LIN {X 0,Y 417.442,Z 383.937,A -85,B 0,C 180,E1 -10178.471,E2 -10178.471} C_VEL
LIN {X 0,Y 417.791,Z 376.994,A -85,B 0,C 180,E1 -10179.929,E2 -10179.929} C_VEL
LIN {X 0,Y 418.22,Z 369.9,A -85,B 0,C 180,E1 -10181.142,E2 -10181.142} C_VEL
LIN {X 0,Y 418.782,Z 361.342,A -85,B 0,C 180,E1 -10182.355,E2 -10182.355} C_VEL
LIN {X 0,Y 419.399,Z 350.75,A -85,B 0,C 180,E1 -10183.568,E2 -10183.568} C_VEL
LIN {X 0,Y 420.122,Z 340.277,A -85,B 0,C 180,E1 -10184.532,E2 -10184.532} C_VEL
LIN {X 0,Y 420.811,Z 328.769,A -85,B 0,C 180,E1 -10185.374,E2 -10185.374} C_VEL
LIN {X 0,Y 421.406,Z 316.866,A -85,B 0,C 180,E1 -10186.035,E2 -10186.035} C_VEL
LIN {X 0,Y 422.047,Z 303.154,A -85,B 0,C 180,E1 -10186.569,E2 -10186.569} C_VEL
LIN {X 0,Y 422.362,Z 290.817,A -85,B 0,C 180,E1 -10186.867,E2 -10186.867} C_VEL
LIN {X 0,Y 422.986,Z 214.349,A -85,B 0,C 180,E1 -10188.185,E2 -10188.185} C_VEL
LIN {X 0,Y 419.308,Z 188.077,A -85,B 0,C 180,E1 -10188.791,E2 -10188.791} C_VEL
LIN {X 0,Y 420.32,Z 170.294,A -85,B 0,C 180,E1 -10192.099,E2 -10192.099} C_VEL
LIN {X 0,Y 421.109,Z 156.698,A -85,B 0,C 180,E1 -10194.66,E2 -10194.66} C_VEL
LIN {X 0,Y 419.458,Z 146.94,A -85,B 0,C 180,E1 -10196.628,E2 -10196.628} C_VEL
LIN {X 0,Y 418.334,Z 141.379,A -85,B 0,C 180,E1 -10197.822,E2 -10197.822} C_VEL
LIN {X 0,Y 418.213,Z 141.391,A -85,B 0,C 180,E1 -10201.396,E2 -10201.396} C_VEL
LIN {X 0,Y 418.267,Z 141.381,A -85,B 0,C 180,E1 -10204.58,E2 -10204.58} C_VEL
LIN {X 0,Y 418.231,Z 141.391,A -85,B 0,C 180,E1 -10207.833,E2 -10207.833} C_VEL
LIN {X 0,Y 418.224,Z 141.385,A -85,B 0,C 180,E1 -10210.948,E2 -10210.948} C_VEL
LIN {X 0,Y 418.211,Z 141.394,A -85,B 0,C 180,E1 -10213.729,E2 -10213.729} C_VEL
LIN {X 0,Y 418.209,Z 141.387,A -85,B 0,C 180,E1 -10216.448,E2 -10216.448} C_VEL
LIN {X 0,Y 418.223,Z 141.387,A -85,B 0,C 180,E1 -10219.13,E2 -10219.13} C_VEL
LIN {X 0,Y 418.226,Z 141.386,A -85,B 0,C 180,E1 -10222.167,E2 -10222.167} C_VEL
LIN {X 0,Y 418.264,Z 141.387,A -85,B 0,C 180,E1 -10225.42,E2 -10225.42} C_VEL
LIN {X 0,Y 418.211,Z 141.387,A -85,B 0,C 180,E1 -10228.604,E2 -10228.604} C_VEL
LIN {X 0,Y 418.292,Z 141.378,A -85,B 0,C 180,E1 -10231.936,E2 -10231.936} C_VEL
LIN {X 0,Y 418.29,Z 141.383,A -85,B 0,C 180,E1 -10235.162,E2 -10235.162} C_VEL
LIN {X 0,Y 418.234,Z 141.384,A -85,B 0,C 180,E1 -10238.303,E2 -10238.303} C_VEL
LIN {X 0,Y 418.276,Z 141.383,A -85,B 0,C 180,E1 -10241.383,E2 -10241.383} C_VEL
LIN {X 0,Y 418.302,Z 141.376,A -85,B 0,C 180,E1 -10244.406,E2 -10244.406} C_VEL
LIN {X 0,Y 418.355,Z 141.371,A -85,B 0,C 180,E1 -10247.385,E2 -10247.385} C_VEL
LIN {X 0,Y 418.339,Z 141.372,A -85,B 0,C 180,E1 -10250.328,E2 -10250.328} C_VEL
LIN {X 0,Y 418.46,Z 141.358,A -85,B 0,C 180,E1 -10253.248,E2 -10253.248} C_VEL
LIN {X 0,Y 418.336,Z 141.374,A -85,B 0,C 180,E1 -10255.181,E2 -10255.181} C_VEL
LIN {X 0,Y 418.543,Z 141.346,A -85,B 0,C 180,E1 -10258.075,E2 -10258.075} C_VEL
LIN {X 0,Y 418.671,Z 141.33,A -85,B 0,C 180,E1 -10260,E2 -10260} C_VEL
LIN {X 0,Y 418.508,Z 141.354,A -85,B 0,C 180,E1 -10262.888,E2 -10262.888} C_VEL
LIN {X 0,Y 418.487,Z 141.357,A -85,B 0,C 180,E1 -10266.751,E2 -10266.751} C_VEL
LIN {X 0,Y 418.34,Z 141.371,A -85,B 0,C 180,E1 -10269.671,E2 -10269.671} C_VEL
LIN {X 0,Y 418.346,Z 141.371,A -85,B 0,C 180,E1 -10273.001,E2 -10273.001} C_VEL
LIN {X 0,Y 418.312,Z 141.377,A -85,B 0,C 180,E1 -10276.735,E2 -10276.735} C_VEL
LIN {X 0,Y 418.27,Z 141.382,A -85,B 0,C 180,E1 -10279.79,E2 -10279.79} C_VEL
LIN {X 0,Y 418.231,Z 141.386,A -85,B 0,C 180,E1 -10282.736,E2 -10282.736} C_VEL
LIN {X 0,Y 418.267,Z 141.385,A -85,B 0,C 180,E1 -10285.904,E2 -10285.904} C_VEL
LIN {X 0,Y 418.264,Z 141.38,A -85,B 0,C 180,E1 -10289.162,E2 -10289.162} C_VEL
LIN {X 0,Y 418.256,Z 141.381,A -85,B 0,C 180,E1 -10292.844,E2 -10292.844} C_VEL
LIN {X 0,Y 418.244,Z 141.386,A -85,B 0,C 180,E1 -10296.238,E2 -10296.238} C_VEL
LIN {X 0,Y 418.253,Z 141.388,A -85,B 0,C 180,E1 -10299.681,E2 -10299.681} C_VEL
LIN {X 0,Y 418.229,Z 141.386,A -85,B 0,C 180,E1 -10302.321,E2 -10302.321} C_VEL
LIN {X 0,Y 418.234,Z 141.385,A -85,B 0,C 180,E1 -10305.109,E2 -10305.109} C_VEL
LIN {X 0,Y 418.239,Z 141.389,A -85,B 0,C 180,E1 -10307.767,E2 -10307.767} C_VEL
LIN {X 0,Y 418.244,Z 141.383,A -85,B 0,C 180,E1 -10310.621,E2 -10310.621} C_VEL
LIN {X 0,Y 418.241,Z 141.385,A -85,B 0,C 180,E1 -10313.976,E2 -10313.976} C_VEL
LIN {X 0,Y 418.256,Z 141.386,A -85,B 0,C 180,E1 -10317.156,E2 -10317.156} C_VEL
LIN {X 0,Y 418.268,Z 141.382,A -85,B 0,C 180,E1 -10320.896,E2 -10320.896} C_VEL
LIN {X 0,Y 418.268,Z 141.38,A -85,B 0,C 180,E1 -10324.096,E2 -10324.096} C_VEL
LIN {X 0,Y 418.232,Z 141.39,A -85,B 0,C 180,E1 -10327.264,E2 -10327.264} C_VEL
LIN {X 0,Y 418.282,Z 141.378,A -85,B 0,C 180,E1 -10330.364,E2 -10330.364} C_VEL
LIN {X 0,Y 418.316,Z 141.376,A -85,B 0,C 180,E1 -10333.405,E2 -10333.405} C_VEL
LIN {X 0,Y 418.346,Z 141.377,A -85,B 0,C 180,E1 -10336.999,E2 -10336.999} C_VEL
LIN {X 0,Y 418.339,Z 141.372,A -85,B 0,C 180,E1 -10340.329,E2 -10340.329} C_VEL
LIN {X 0,Y 418.46,Z 141.358,A -85,B 0,C 180,E1 -10343.249,E2 -10343.249} C_VEL
LIN {X 0,Y 418.336,Z 141.377,A -85,B 0,C 180,E1 -10345.182,E2 -10345.182} C_VEL
LIN {X 0,Y 418.543,Z 141.351,A -85,B 0,C 180,E1 -10348.076,E2 -10348.076} C_VEL
LIN {X 0,Y 418.534,Z 141.54,A -85,B 0,C 180,E1 -10348.797,E2 -10348.797} C_VEL
LIN {X 0,Y 419.76,Z 148.679,A -85,B 0,C 180,E1 -10350.48,E2 -10350.48} C_VEL
LIN {X 0,Y 419.846,Z 152.338,A -85,B 0,C 180,E1 -10351.31,E2 -10351.31} C_VEL
LIN {X 0,Y 423.514,Z 171.824,A -85,B 0,C 180,E1 -10351.804,E2 -10351.804} C_VEL
LIN {X 0,Y 423.009,Z 213.686,A -85,B 0,C 180,E1 -10352.52,E2 -10352.52} C_VEL
LIN {X 0,Y 422.295,Z 219.534,A -85,B 0,C 180,E1 -10352.597,E2 -10352.597} C_VEL
LIN {X 0,Y 416.394,Z 238.495,A -85,B 0,C 180,E1 -10352.713,E2 -10352.713} C_VEL
LIN {X 0,Y 415.758,Z 244.339,A -85,B 0,C 180,E1 -10352.794,E2 -10352.794} C_VEL
LIN {X 0,Y 415.479,Z 262.827,A -85,B 0,C 180,E1 -10353.167,E2 -10353.167} C_VEL
LIN {X 0,Y 415.18,Z 275.079,A -85,B 0,C 180,E1 -10353.598,E2 -10353.598} C_VEL
LIN {X 0,Y 414.746,Z 286.827,A -85,B 0,C 180,E1 -10354.191,E2 -10354.191} C_VEL
LIN {X 0,Y 414.175,Z 298.648,A -85,B 0,C 180,E1 -10354.989,E2 -10354.989} C_VEL
LIN {X 0,Y 413.529,Z 310.039,A -85,B 0,C 180,E1 -10355.975,E2 -10355.975} C_VEL
LIN {X 0,Y 412.809,Z 320.326,A -85,B 0,C 180,E1 -10357.09,E2 -10357.09} C_VEL
LIN {X 0,Y 412.06,Z 330.114,A -85,B 0,C 180,E1 -10358.416,E2 -10358.416} C_VEL
LIN {X 0,Y 411.453,Z 338.576,A -85,B 0,C 180,E1 -10359.835,E2 -10359.835} C_VEL
LIN {X 0,Y 410.99,Z 345.766,A -85,B 0,C 180,E1 -10361.341,E2 -10361.341} C_VEL
LIN {X 0,Y 410.619,Z 351.496,A -85,B 0,C 180,E1 -10362.856,E2 -10362.856} C_VEL
LIN {X 0,Y 410.329,Z 355.996,A -85,B 0,C 180,E1 -10364.38,E2 -10364.38} C_VEL
LIN {X 0,Y 410.103,Z 359.379,A -85,B 0,C 180,E1 -10365.914,E2 -10365.914} C_VEL
LIN {X 0,Y 409.981,Z 361.058,A -85,B 0,C 180,E1 -10366.943,E2 -10366.943} C_VEL
LIN {X 0,Y 409.908,Z 362.294,A -85,B 0,C 180,E1 -10367.976,E2 -10367.976} C_VEL
LIN {X 0,Y 409.918,Z 363.263,A -85,B 0,C 180,E1 -10369.444,E2 -10369.444} C_VEL
LIN {X 0,Y 409.88,Z 363.307,A -85,B 0,C 180,E1 -10371.105,E2 -10371.105} C_VEL
LIN {X 0,Y 409.945,Z 362.679,A -85,B 0,C 180,E1 -10372.217,E2 -10372.217} C_VEL
LIN {X 0,Y 410.041,Z 361.707,A -85,B 0,C 180,E1 -10373.217,E2 -10373.217} C_VEL
LIN {X 0,Y 410.288,Z 359.319,A -85,B 0,C 180,E1 -10374.789,E2 -10374.789} C_VEL
LIN {X 0,Y 410.566,Z 355.675,A -85,B 0,C 180,E1 -10376.428,E2 -10376.428} C_VEL
LIN {X 0,Y 410.96,Z 350.746,A -85,B 0,C 180,E1 -10378.053,E2 -10378.053} C_VEL
LIN {X 0,Y 411.519,Z 344.278,A -85,B 0,C 180,E1 -10379.688,E2 -10379.688} C_VEL
LIN {X 0,Y 412.226,Z 336.472,A -85,B 0,C 180,E1 -10381.248,E2 -10381.248} C_VEL
LIN {X 0,Y 413.047,Z 327.312,A -85,B 0,C 180,E1 -10382.699,E2 -10382.699} C_VEL
LIN {X 0,Y 413.821,Z 317.593,A -85,B 0,C 180,E1 -10383.941,E2 -10383.941} C_VEL
LIN {X 0,Y 414.737,Z 306.944,A -85,B 0,C 180,E1 -10385.032,E2 -10385.032} C_VEL
LIN {X 0,Y 415.542,Z 296.131,A -85,B 0,C 180,E1 -10385.91,E2 -10385.91} C_VEL
LIN {X 0,Y 416.147,Z 283.863,A -85,B 0,C 180,E1 -10386.686,E2 -10386.686} C_VEL
LIN {X 0,Y 416.694,Z 271.1,A -85,B 0,C 180,E1 -10387.272,E2 -10387.272} C_VEL
LIN {X 0,Y 417.018,Z 257.825,A -85,B 0,C 180,E1 -10387.664,E2 -10387.664} C_VEL
LIN {X 0,Y 418.238,Z 172.5,A -85,B 0,C 180,E1 -10389.181,E2 -10389.181} C_VEL
LIN {X 0,Y 414.446,Z 156.312,A -85,B 0,C 180,E1 -10389.696,E2 -10389.696} C_VEL
LIN {X 0,Y 413.397,Z 153.147,A -85,B 0,C 180,E1 -10389.83,E2 -10389.83} C_VEL
LIN {X 0,Y 411.182,Z 142.299,A -85,B 0,C 180,E1 -10392.548,E2 -10392.548} C_VEL
LIN {X 0,Y 411.164,Z 142.275,A -85,B 0,C 180,E1 -10395.882,E2 -10395.882} C_VEL
LIN {X 0,Y 411.158,Z 142.269,A -85,B 0,C 180,E1 -10399.493,E2 -10399.493} C_VEL
LIN {X 0,Y 411.186,Z 142.266,A -85,B 0,C 180,E1 -10402.026,E2 -10402.026} C_VEL
LIN {X 0,Y 411.203,Z 142.267,A -85,B 0,C 180,E1 -10405.124,E2 -10405.124} C_VEL
LIN {X 0,Y 411.16,Z 142.269,A -85,B 0,C 180,E1 -10408.002,E2 -10408.002} C_VEL
LIN {X 0,Y 411.17,Z 142.267,A -85,B 0,C 180,E1 -10411.407,E2 -10411.407} C_VEL
LIN {X 0,Y 411.187,Z 142.268,A -85,B 0,C 180,E1 -10414.942,E2 -10414.942} C_VEL
LIN {X 0,Y 411.196,Z 142.259,A -85,B 0,C 180,E1 -10417.913,E2 -10417.913} C_VEL
LIN {X 0,Y 411.178,Z 142.262,A -85,B 0,C 180,E1 -10421.049,E2 -10421.049} C_VEL
LIN {X 0,Y 411.195,Z 142.264,A -85,B 0,C 180,E1 -10424.13,E2 -10424.13} C_VEL
LIN {X 0,Y 411.296,Z 142.25,A -85,B 0,C 180,E1 -10427.166,E2 -10427.166} C_VEL
LIN {X 0,Y 411.274,Z 142.252,A -85,B 0,C 180,E1 -10430.161,E2 -10430.161} C_VEL
LIN {X 0,Y 411.391,Z 142.232,A -85,B 0,C 180,E1 -10433.132,E2 -10433.132} C_VEL
LIN {X 0,Y 411.284,Z 142.249,A -85,B 0,C 180,E1 -10435.099,E2 -10435.099} C_VEL
LIN {X 0,Y 411.502,Z 142.22,A -85,B 0,C 180,E1 -10438.043,E2 -10438.043} C_VEL
LIN {X 0,Y 411.377,Z 142.238,A -85,B 0,C 180,E1 -10440.979,E2 -10440.979} C_VEL
LIN {X 0,Y 411.428,Z 142.225,A -85,B 0,C 180,E1 -10442.938,E2 -10442.938} C_VEL
LIN {X 0,Y 411.429,Z 142.235,A -85,B 0,C 180,E1 -10445.883,E2 -10445.883} C_VEL
LIN {X 0,Y 411.312,Z 142.243,A -85,B 0,C 180,E1 -10448.846,E2 -10448.846} C_VEL
LIN {X 0,Y 411.284,Z 142.248,A -85,B 0,C 180,E1 -10451.833,E2 -10451.833} C_VEL
LIN {X 0,Y 411.256,Z 142.254,A -85,B 0,C 180,E1 -10454.853,E2 -10454.853} C_VEL
LIN {X 0,Y 411.245,Z 142.251,A -85,B 0,C 180,E1 -10457.916,E2 -10457.916} C_VEL
LIN {X 0,Y 411.198,Z 142.264,A -85,B 0,C 180,E1 -10461.034,E2 -10461.034} C_VEL
LIN {X 0,Y 411.219,Z 142.258,A -85,B 0,C 180,E1 -10464.216,E2 -10464.216} C_VEL
LIN {X 0,Y 411.181,Z 142.265,A -85,B 0,C 180,E1 -10467.484,E2 -10467.484} C_VEL
LIN {X 0,Y 411.199,Z 142.259,A -85,B 0,C 180,E1 -10469.713,E2 -10469.713} C_VEL
LIN {X 0,Y 411.209,Z 142.261,A -85,B 0,C 180,E1 -10473.156,E2 -10473.156} C_VEL
LIN {X 0,Y 411.194,Z 142.267,A -85,B 0,C 180,E1 -10476.552,E2 -10476.552} C_VEL
LIN {X 0,Y 411.18,Z 142.265,A -85,B 0,C 180,E1 -10479.722,E2 -10479.722} C_VEL
LIN {X 0,Y 411.172,Z 142.267,A -85,B 0,C 180,E1 -10483.134,E2 -10483.134} C_VEL
LIN {X 0,Y 411.17,Z 142.268,A -85,B 0,C 180,E1 -10485.881,E2 -10485.881} C_VEL
LIN {X 0,Y 411.163,Z 142.272,A -85,B 0,C 180,E1 -10488.772,E2 -10488.772} C_VEL
LIN {X 0,Y 411.192,Z 142.262,A -85,B 0,C 180,E1 -10492.026,E2 -10492.026} C_VEL
LIN {X 0,Y 411.208,Z 142.259,A -85,B 0,C 180,E1 -10495.666,E2 -10495.666} C_VEL
LIN {X 0,Y 411.192,Z 142.268,A -85,B 0,C 180,E1 -10499.152,E2 -10499.152} C_VEL
LIN {X 0,Y 411.255,Z 142.294,A -85,B 0,C 180,E1 -10501.05,E2 -10501.05} C_VEL
LIN {X 0,Y 413.993,Z 154.656,A -85,B 0,C 180,E1 -10503.808,E2 -10503.808} C_VEL
LIN {X 0,Y 414.854,Z 159.972,A -85,B 0,C 180,E1 -10504.943,E2 -10504.943} C_VEL
LIN {X 0,Y 413.792,Z 174.576,A -85,B 0,C 180,E1 -10507.796,E2 -10507.796} C_VEL
LIN {X 0,Y 412.989,Z 187.099,A -85,B 0,C 180,E1 -10510.206,E2 -10510.206} C_VEL
LIN {X 0,Y 417.154,Z 211.973,A -85,B 0,C 180,E1 -10510.896,E2 -10510.896} C_VEL
LIN {X 0,Y 417.661,Z 218.162,A -85,B 0,C 180,E1 -10511.037,E2 -10511.037} C_VEL
LIN {X 0,Y 416.649,Z 296.536,A -85,B 0,C 180,E1 -10512.451,E2 -10512.451} C_VEL
LIN {X 0,Y 416.008,Z 309.504,A -85,B 0,C 180,E1 -10512.867,E2 -10512.867} C_VEL
LIN {X 0,Y 415.3,Z 322.073,A -85,B 0,C 180,E1 -10513.47,E2 -10513.47} C_VEL
LIN {X 0,Y 414.419,Z 334.091,A -85,B 0,C 180,E1 -10514.256,E2 -10514.256} C_VEL
LIN {X 0,Y 413.529,Z 345.578,A -85,B 0,C 180,E1 -10515.231,E2 -10515.231} C_VEL
LIN {X 0,Y 412.662,Z 355.955,A -85,B 0,C 180,E1 -10516.331,E2 -10516.331} C_VEL
LIN {X 0,Y 412.017,Z 364.46,A -85,B 0,C 180,E1 -10517.439,E2 -10517.439} C_VEL
LIN {X 0,Y 411.217,Z 373.705,A -85,B 0,C 180,E1 -10518.914,E2 -10518.914} C_VEL
LIN {X 0,Y 410.654,Z 381.157,A -85,B 0,C 180,E1 -10520.394,E2 -10520.394} C_VEL
LIN {X 0,Y 410.266,Z 388.053,A -85,B 0,C 180,E1 -10522.123,E2 -10522.123} C_VEL
LIN {X 0,Y 410.044,Z 393.055,A -85,B 0,C 180,E1 -10523.775,E2 -10523.775} C_VEL
LIN {X 0,Y 410.009,Z 396.102,A -85,B 0,C 180,E1 -10525.083,E2 -10525.083} C_VEL
LIN {X 0,Y 409.971,Z 399.185,A -85,B 0,C 180,E1 -10527.052,E2 -10527.052} C_VEL
LIN {X 0,Y 410.019,Z 400.129,A -85,B 0,C 180,E1 -10528.035,E2 -10528.035} C_VEL
LIN {X 0,Y 409.982,Z 400.664,A -85,B 0,C 180,E1 -10529.018,E2 -10529.018} C_VEL
LIN {X 0,Y 409.979,Z 400.766,A -85,B 0,C 180,E1 -10530,E2 -10530} C_VEL
LIN {X 0,Y 410.021,Z 399.803,A -85,B 0,C 180,E1 -10531.964,E2 -10531.964} C_VEL
LIN {X 0,Y 409.99,Z 398.717,A -85,B 0,C 180,E1 -10532.948,E2 -10532.948} C_VEL
LIN {X 0,Y 409.944,Z 397.171,A -85,B 0,C 180,E1 -10533.932,E2 -10533.932} C_VEL
LIN {X 0,Y 409.997,Z 394.061,A -85,B 0,C 180,E1 -10535.41,E2 -10535.41} C_VEL
LIN {X 0,Y 410.078,Z 389.873,A -85,B 0,C 180,E1 -10536.89,E2 -10536.89} C_VEL
LIN {X 0,Y 410.368,Z 383.477,A -85,B 0,C 180,E1 -10538.618,E2 -10538.618} C_VEL
LIN {X 0,Y 410.731,Z 376.502,A -85,B 0,C 180,E1 -10540.101,E2 -10540.101} C_VEL
LIN {X 0,Y 411.323,Z 367.744,A -85,B 0,C 180,E1 -10541.581,E2 -10541.581} C_VEL
LIN {X 0,Y 411.907,Z 358.756,A -85,B 0,C 180,E1 -10542.815,E2 -10542.815} C_VEL
LIN {X 0,Y 412.523,Z 348.873,A -85,B 0,C 180,E1 -10543.924,E2 -10543.924} C_VEL
LIN {X 0,Y 413.3,Z 338.012,A -85,B 0,C 180,E1 -10544.903,E2 -10544.903} C_VEL
LIN {X 0,Y 414.029,Z 325.801,A -85,B 0,C 180,E1 -10545.759,E2 -10545.759} C_VEL
LIN {X 0,Y 414.709,Z 313.047,A -85,B 0,C 180,E1 -10546.427,E2 -10546.427} C_VEL
LIN {X 0,Y 415.307,Z 300.463,A -85,B 0,C 180,E1 -10546.877,E2 -10546.877} C_VEL
LIN {X 0,Y 415.557,Z 284.461,A -85,B 0,C 180,E1 -10547.215,E2 -10547.215} C_VEL
LIN {X 0,Y 416.168,Z 215.226,A -85,B 0,C 180,E1 -10548.426,E2 -10548.426} C_VEL
LIN {X 0,Y 412.372,Z 187.703,A -85,B 0,C 180,E1 -10549.087,E2 -10549.087} C_VEL
LIN {X 0,Y 413.612,Z 167.046,A -85,B 0,C 180,E1 -10553.005,E2 -10553.005} C_VEL
LIN {X 0,Y 414.141,Z 157.479,A -85,B 0,C 180,E1 -10554.835,E2 -10554.835} C_VEL
LIN {X 0,Y 411.825,Z 144.813,A -85,B 0,C 180,E1 -10557.45,E2 -10557.45} C_VEL
LIN {X 0,Y 411.29,Z 142.256,A -85,B 0,C 180,E1 -10558.028,E2 -10558.028} C_VEL
LIN {X 0,Y 411.184,Z 142.267,A -85,B 0,C 180,E1 -10561.283,E2 -10561.283} C_VEL
LIN {X 0,Y 411.207,Z 142.262,A -85,B 0,C 180,E1 -10564.333,E2 -10564.333} C_VEL
LIN {X 0,Y 411.198,Z 142.266,A -85,B 0,C 180,E1 -10567.973,E2 -10567.973} C_VEL
LIN {X 0,Y 411.184,Z 142.263,A -85,B 0,C 180,E1 -10570.504,E2 -10570.504} C_VEL
LIN {X 0,Y 411.174,Z 142.264,A -85,B 0,C 180,E1 -10573.133,E2 -10573.133} C_VEL
LIN {X 0,Y 411.168,Z 142.269,A -85,B 0,C 180,E1 -10575.881,E2 -10575.881} C_VEL
LIN {X 0,Y 411.164,Z 142.265,A -85,B 0,C 180,E1 -10578.771,E2 -10578.771} C_VEL
LIN {X 0,Y 411.192,Z 142.263,A -85,B 0,C 180,E1 -10582.026,E2 -10582.026} C_VEL
LIN {X 0,Y 411.205,Z 142.264,A -85,B 0,C 180,E1 -10585.666,E2 -10585.666} C_VEL
LIN {X 0,Y 411.19,Z 142.266,A -85,B 0,C 180,E1 -10589.152,E2 -10589.152} C_VEL
LIN {X 0,Y 411.259,Z 142.253,A -85,B 0,C 180,E1 -10592.522,E2 -10592.522} C_VEL
LIN {X 0,Y 411.22,Z 142.259,A -85,B 0,C 180,E1 -10595.784,E2 -10595.784} C_VEL
LIN {X 0,Y 411.197,Z 142.265,A -85,B 0,C 180,E1 -10598.966,E2 -10598.966} C_VEL
LIN {X 0,Y 411.246,Z 142.254,A -85,B 0,C 180,E1 -10602.084,E2 -10602.084} C_VEL
LIN {X 0,Y 411.26,Z 142.258,A -85,B 0,C 180,E1 -10605.147,E2 -10605.147} C_VEL
LIN {X 0,Y 411.284,Z 142.25,A -85,B 0,C 180,E1 -10608.167,E2 -10608.167} C_VEL
LIN {X 0,Y 411.319,Z 142.249,A -85,B 0,C 180,E1 -10611.154,E2 -10611.154} C_VEL
LIN {X 0,Y 411.444,Z 142.23,A -85,B 0,C 180,E1 -10614.117,E2 -10614.117} C_VEL
LIN {X 0,Y 411.512,Z 142.222,A -85,B 0,C 180,E1 -10618.042,E2 -10618.042} C_VEL
LIN {X 0,Y 411.64,Z 142.206,A -85,B 0,C 180,E1 -10620,E2 -10620} C_VEL
LIN {X 0,Y 411.464,Z 142.231,A -85,B 0,C 180,E1 -10622.937,E2 -10622.937} C_VEL
LIN {X 0,Y 411.451,Z 142.232,A -85,B 0,C 180,E1 -10626.867,E2 -10626.867} C_VEL
LIN {X 0,Y 411.292,Z 142.25,A -85,B 0,C 180,E1 -10629.839,E2 -10629.839} C_VEL
LIN {X 0,Y 411.305,Z 142.248,A -85,B 0,C 180,E1 -10633.104,E2 -10633.104} C_VEL
LIN {X 0,Y 411.257,Z 142.254,A -85,B 0,C 180,E1 -10636.889,E2 -10636.889} C_VEL
LIN {X 0,Y 411.23,Z 142.261,A -85,B 0,C 180,E1 -10639.987,E2 -10639.987} C_VEL
LIN {X 0,Y 411.195,Z 142.261,A -85,B 0,C 180,E1 -10643.148,E2 -10643.148} C_VEL
LIN {X 0,Y 411.236,Z 142.259,A -85,B 0,C 180,E1 -10646.381,E2 -10646.381} C_VEL
LIN {X 0,Y 411.199,Z 142.264,A -85,B 0,C 180,E1 -10649.713,E2 -10649.713} C_VEL
LIN {X 0,Y 411.205,Z 142.26,A -85,B 0,C 180,E1 -10653.156,E2 -10653.156} C_VEL
LIN {X 0,Y 411.191,Z 142.262,A -85,B 0,C 180,E1 -10656.553,E2 -10656.553} C_VEL
LIN {X 0,Y 411.217,Z 142.265,A -85,B 0,C 180,E1 -10659.729,E2 -10659.729} C_VEL
LIN {X 0,Y 411.172,Z 142.265,A -85,B 0,C 180,E1 -10663.134,E2 -10663.134} C_VEL
LIN {X 0,Y 411.166,Z 142.269,A -85,B 0,C 180,E1 -10665.881,E2 -10665.881} C_VEL
LIN {X 0,Y 411.162,Z 142.265,A -85,B 0,C 180,E1 -10668.772,E2 -10668.772} C_VEL
LIN {X 0,Y 411.19,Z 142.263,A -85,B 0,C 180,E1 -10672.026,E2 -10672.026} C_VEL
LIN {X 0,Y 411.203,Z 142.264,A -85,B 0,C 180,E1 -10675.666,E2 -10675.666} C_VEL
LIN {X 0,Y 411.189,Z 142.266,A -85,B 0,C 180,E1 -10679.153,E2 -10679.153} C_VEL
LIN {X 0,Y 411.258,Z 142.253,A -85,B 0,C 180,E1 -10682.522,E2 -10682.522} C_VEL
LIN {X 0,Y 411.219,Z 142.259,A -85,B 0,C 180,E1 -10685.784,E2 -10685.784} C_VEL
LIN {X 0,Y 411.196,Z 142.266,A -85,B 0,C 180,E1 -10688.966,E2 -10688.966} C_VEL
LIN {X 0,Y 411.245,Z 142.255,A -85,B 0,C 180,E1 -10692.085,E2 -10692.085} C_VEL
LIN {X 0,Y 411.259,Z 142.258,A -85,B 0,C 180,E1 -10695.148,E2 -10695.148} C_VEL
LIN {X 0,Y 411.283,Z 142.25,A -85,B 0,C 180,E1 -10698.167,E2 -10698.167} C_VEL
LIN {X 0,Y 411.319,Z 142.249,A -85,B 0,C 180,E1 -10701.154,E2 -10701.154} C_VEL
LIN {X 0,Y 411.444,Z 142.231,A -85,B 0,C 180,E1 -10704.118,E2 -10704.118} C_VEL
LIN {X 0,Y 411.512,Z 142.227,A -85,B 0,C 180,E1 -10708.043,E2 -10708.043} C_VEL
LIN {X 0,Y 411.489,Z 142.365,A -85,B 0,C 180,E1 -10708.593,E2 -10708.593} C_VEL
LIN {X 0,Y 412.843,Z 150.275,A -85,B 0,C 180,E1 -10710.488,E2 -10710.488} C_VEL
LIN {X 0,Y 412.928,Z 152.724,A -85,B 0,C 180,E1 -10711.032,E2 -10711.032} C_VEL
LIN {X 0,Y 416.688,Z 173.001,A -85,B 0,C 180,E1 -10711.555,E2 -10711.555} C_VEL
LIN {X 0,Y 415.758,Z 244.339,A -85,B 0,C 180,E1 -10712.794,E2 -10712.794} C_VEL
LIN {X 0,Y 415.439,Z 248.253,A -85,B 0,C 180,E1 -10712.85,E2 -10712.85} C_VEL
LIN {X 0,Y 413.316,Z 255.899,A -85,B 0,C 180,E1 -10712.913,E2 -10712.913} C_VEL
LIN {X 0,Y 409.135,Z 268.076,A -85,B 0,C 180,E1 -10713.1,E2 -10713.1} C_VEL
LIN {X 0,Y 408.368,Z 272.839,A -85,B 0,C 180,E1 -10713.253,E2 -10713.253} C_VEL
LIN {X 0,Y 408.312,Z 274.666,A -85,B 0,C 180,E1 -10713.329,E2 -10713.329} C_VEL
LIN {X 0,Y 407.854,Z 286.988,A -85,B 0,C 180,E1 -10713.953,E2 -10713.953} C_VEL
LIN {X 0,Y 407.295,Z 298.053,A -85,B 0,C 180,E1 -10714.702,E2 -10714.702} C_VEL
LIN {X 0,Y 406.62,Z 309.609,A -85,B 0,C 180,E1 -10715.704,E2 -10715.704} C_VEL
LIN {X 0,Y 405.886,Z 320.05,A -85,B 0,C 180,E1 -10716.837,E2 -10716.837} C_VEL
LIN {X 0,Y 405.21,Z 328.586,A -85,B 0,C 180,E1 -10717.976,E2 -10717.976} C_VEL
LIN {X 0,Y 404.633,Z 336.423,A -85,B 0,C 180,E1 -10719.245,E2 -10719.245} C_VEL
LIN {X 0,Y 404.072,Z 344.087,A -85,B 0,C 180,E1 -10720.776,E2 -10720.776} C_VEL
LIN {X 0,Y 403.633,Z 350.609,A -85,B 0,C 180,E1 -10722.417,E2 -10722.417} C_VEL
LIN {X 0,Y 403.299,Z 355.81,A -85,B 0,C 180,E1 -10724.121,E2 -10724.121} C_VEL
LIN {X 0,Y 403.053,Z 359.334,A -85,B 0,C 180,E1 -10725.681,E2 -10725.681} C_VEL
LIN {X 0,Y 402.863,Z 361.808,A -85,B 0,C 180,E1 -10727.252,E2 -10727.252} C_VEL
LIN {X 0,Y 402.803,Z 362.878,A -85,B 0,C 180,E1 -10728.304,E2 -10728.304} C_VEL
LIN {X 0,Y 402.822,Z 363.626,A -85,B 0,C 180,E1 -10729.588,E2 -10729.588} C_VEL
LIN {X 0,Y 402.829,Z 363.485,A -85,B 0,C 180,E1 -10731.493,E2 -10731.493} C_VEL
LIN {X 0,Y 402.879,Z 362.797,A -85,B 0,C 180,E1 -10732.568,E2 -10732.568} C_VEL
LIN {X 0,Y 403.033,Z 361.643,A -85,B 0,C 180,E1 -10733.645,E2 -10733.645} C_VEL
LIN {X 0,Y 403.262,Z 359.485,A -85,B 0,C 180,E1 -10735.008,E2 -10735.008} C_VEL
LIN {X 0,Y 403.492,Z 356.523,A -85,B 0,C 180,E1 -10736.37,E2 -10736.37} C_VEL
LIN {X 0,Y 403.892,Z 351.785,A -85,B 0,C 180,E1 -10738.023,E2 -10738.023} C_VEL
LIN {X 0,Y 404.484,Z 345.544,A -85,B 0,C 180,E1 -10739.685,E2 -10739.685} C_VEL
LIN {X 0,Y 405.232,Z 337.515,A -85,B 0,C 180,E1 -10741.352,E2 -10741.352} C_VEL
LIN {X 0,Y 406.036,Z 329.138,A -85,B 0,C 180,E1 -10742.745,E2 -10742.745} C_VEL
LIN {X 0,Y 406.909,Z 319.272,A -85,B 0,C 180,E1 -10744.062,E2 -10744.062} C_VEL
LIN {X 0,Y 407.89,Z 308.066,A -85,B 0,C 180,E1 -10745.255,E2 -10745.255} C_VEL
LIN {X 0,Y 408.788,Z 296.879,A -85,B 0,C 180,E1 -10746.192,E2 -10746.192} C_VEL
LIN {X 0,Y 409.46,Z 284.345,A -85,B 0,C 180,E1 -10747,E2 -10747} C_VEL
LIN {X 0,Y 410.018,Z 271.622,A -85,B 0,C 180,E1 -10747.597,E2 -10747.597} C_VEL
LIN {X 0,Y 410.38,Z 258.105,A -85,B 0,C 180,E1 -10748.003,E2 -10748.003} C_VEL
LIN {X 0,Y 411.742,Z 173.912,A -85,B 0,C 180,E1 -10749.521,E2 -10749.521} C_VEL
LIN {X 0,Y 408.264,Z 158.893,A -85,B 0,C 180,E1 -10750.015,E2 -10750.015} C_VEL
LIN {X 0,Y 406.313,Z 153.449,A -85,B 0,C 180,E1 -10750.263,E2 -10750.263} C_VEL
LIN {X 0,Y 404.12,Z 143.149,A -85,B 0,C 180,E1 -10752.913,E2 -10752.913} C_VEL
LIN {X 0,Y 404.144,Z 143.15,A -85,B 0,C 180,E1 -10755.926,E2 -10755.926} C_VEL
LIN {X 0,Y 404.102,Z 143.153,A -85,B 0,C 180,E1 -10758.633,E2 -10758.633} C_VEL
LIN {X 0,Y 404.14,Z 143.146,A -85,B 0,C 180,E1 -10761.495,E2 -10761.495} C_VEL
LIN {X 0,Y 404.174,Z 143.14,A -85,B 0,C 180,E1 -10764.983,E2 -10764.983} C_VEL
LIN {X 0,Y 404.134,Z 143.146,A -85,B 0,C 180,E1 -10768.444,E2 -10768.444} C_VEL
LIN {X 0,Y 404.148,Z 143.144,A -85,B 0,C 180,E1 -10770.863,E2 -10770.863} C_VEL
LIN {X 0,Y 404.152,Z 143.143,A -85,B 0,C 180,E1 -10774.724,E2 -10774.724} C_VEL
LIN {X 0,Y 404.163,Z 143.134,A -85,B 0,C 180,E1 -10777.508,E2 -10777.508} C_VEL
LIN {X 0,Y 404.131,Z 143.141,A -85,B 0,C 180,E1 -10780.706,E2 -10780.706} C_VEL
LIN {X 0,Y 404.171,Z 143.139,A -85,B 0,C 180,E1 -10783.846,E2 -10783.846} C_VEL
LIN {X 0,Y 404.265,Z 143.126,A -85,B 0,C 180,E1 -10786.938,E2 -10786.938} C_VEL
LIN {X 0,Y 404.242,Z 143.125,A -85,B 0,C 180,E1 -10789.988,E2 -10789.988} C_VEL
LIN {X 0,Y 404.341,Z 143.11,A -85,B 0,C 180,E1 -10793.012,E2 -10793.012} C_VEL
LIN {X 0,Y 404.255,Z 143.125,A -85,B 0,C 180,E1 -10795.013,E2 -10795.013} C_VEL
LIN {X 0,Y 404.471,Z 143.095,A -85,B 0,C 180,E1 -10798.009,E2 -10798.009} C_VEL
LIN {X 0,Y 404.348,Z 143.114,A -85,B 0,C 180,E1 -10800.996,E2 -10800.996} C_VEL
LIN {X 0,Y 404.387,Z 143.101,A -85,B 0,C 180,E1 -10802.989,E2 -10802.989} C_VEL
LIN {X 0,Y 404.378,Z 143.112,A -85,B 0,C 180,E1 -10805.986,E2 -10805.986} C_VEL
LIN {X 0,Y 404.261,Z 143.122,A -85,B 0,C 180,E1 -10809.002,E2 -10809.002} C_VEL
LIN {X 0,Y 404.257,Z 143.122,A -85,B 0,C 180,E1 -10812.042,E2 -10812.042} C_VEL
LIN {X 0,Y 404.203,Z 143.135,A -85,B 0,C 180,E1 -10815.118,E2 -10815.118} C_VEL
LIN {X 0,Y 404.205,Z 143.127,A -85,B 0,C 180,E1 -10818.239,E2 -10818.239} C_VEL
LIN {X 0,Y 404.141,Z 143.137,A -85,B 0,C 180,E1 -10821.42,E2 -10821.42} C_VEL
LIN {X 0,Y 404.169,Z 143.139,A -85,B 0,C 180,E1 -10824.666,E2 -10824.666} C_VEL
LIN {X 0,Y 404.122,Z 143.142,A -85,B 0,C 180,E1 -10828.005,E2 -10828.005} C_VEL
LIN {X 0,Y 404.146,Z 143.138,A -85,B 0,C 180,E1 -10830.285,E2 -10830.285} C_VEL
LIN {X 0,Y 404.147,Z 143.137,A -85,B 0,C 180,E1 -10833.812,E2 -10833.812} C_VEL
LIN {X 0,Y 404.137,Z 143.142,A -85,B 0,C 180,E1 -10836.875,E2 -10836.875} C_VEL
LIN {X 0,Y 404.12,Z 143.146,A -85,B 0,C 180,E1 -10840.075,E2 -10840.075} C_VEL
LIN {X 0,Y 404.152,Z 143.141,A -85,B 0,C 180,E1 -10843.083,E2 -10843.083} C_VEL
LIN {X 0,Y 404.15,Z 143.142,A -85,B 0,C 180,E1 -10845.926,E2 -10845.926} C_VEL
LIN {X 0,Y 404.117,Z 143.151,A -85,B 0,C 180,E1 -10848.634,E2 -10848.634} C_VEL
LIN {X 0,Y 404.15,Z 143.142,A -85,B 0,C 180,E1 -10851.493,E2 -10851.493} C_VEL
LIN {X 0,Y 404.187,Z 143.133,A -85,B 0,C 180,E1 -10854.984,E2 -10854.984} C_VEL
LIN {X 0,Y 404.145,Z 143.147,A -85,B 0,C 180,E1 -10858.554,E2 -10858.554} C_VEL
LIN {X 0,Y 404.21,Z 143.24,A -85,B 0,C 180,E1 -10860.697,E2 -10860.697} C_VEL
LIN {X 0,Y 406.783,Z 154.619,A -85,B 0,C 180,E1 -10863.307,E2 -10863.307} C_VEL
LIN {X 0,Y 407.967,Z 161.266,A -85,B 0,C 180,E1 -10864.763,E2 -10864.763} C_VEL
LIN {X 0,Y 407.438,Z 168.655,A -85,B 0,C 180,E1 -10866.239,E2 -10866.239} C_VEL
LIN {X 0,Y 406.144,Z 186.704,A -85,B 0,C 180,E1 -10869.795,E2 -10869.795} C_VEL
LIN {X 0,Y 410.364,Z 211.552,A -85,B 0,C 180,E1 -10870.519,E2 -10870.519} C_VEL
LIN {X 0,Y 411.047,Z 218.44,A -85,B 0,C 180,E1 -10870.686,E2 -10870.686} C_VEL
LIN {X 0,Y 410,Z 295.498,A -85,B 0,C 180,E1 -10872.093,E2 -10872.093} C_VEL
LIN {X 0,Y 409.359,Z 308.693,A -85,B 0,C 180,E1 -10872.515,E2 -10872.515} C_VEL
LIN {X 0,Y 408.604,Z 321.385,A -85,B 0,C 180,E1 -10873.127,E2 -10873.127} C_VEL
LIN {X 0,Y 407.757,Z 332.708,A -85,B 0,C 180,E1 -10873.863,E2 -10873.863} C_VEL
LIN {X 0,Y 406.754,Z 344.396,A -85,B 0,C 180,E1 -10874.851,E2 -10874.851} C_VEL
LIN {X 0,Y 405.855,Z 354.918,A -85,B 0,C 180,E1 -10875.97,E2 -10875.97} C_VEL
LIN {X 0,Y 405.066,Z 364.429,A -85,B 0,C 180,E1 -10877.219,E2 -10877.219} C_VEL
LIN {X 0,Y 404.204,Z 373.606,A -85,B 0,C 180,E1 -10878.72,E2 -10878.72} C_VEL
LIN {X 0,Y 403.614,Z 381.018,A -85,B 0,C 180,E1 -10880.225,E2 -10880.225} C_VEL
LIN {X 0,Y 403.202,Z 387.863,A -85,B 0,C 180,E1 -10881.984,E2 -10881.984} C_VEL
LIN {X 0,Y 402.934,Z 393.241,A -85,B 0,C 180,E1 -10883.827,E2 -10883.827} C_VEL
LIN {X 0,Y 402.918,Z 395.855,A -85,B 0,C 180,E1 -10884.996,E2 -10884.996} C_VEL
LIN {X 0,Y 402.87,Z 398.904,A -85,B 0,C 180,E1 -10887,E2 -10887} C_VEL
LIN {X 0,Y 402.947,Z 399.837,A -85,B 0,C 180,E1 -10888.001,E2 -10888.001} C_VEL
LIN {X 0,Y 402.907,Z 400.346,A -85,B 0,C 180,E1 -10889,E2 -10889} C_VEL
LIN {X 0,Y 402.901,Z 400.435,A -85,B 0,C 180,E1 -10890,E2 -10890} C_VEL
LIN {X 0,Y 402.95,Z 399.448,A -85,B 0,C 180,E1 -10891.999,E2 -10891.999} C_VEL
LIN {X 0,Y 402.89,Z 398.338,A -85,B 0,C 180,E1 -10893,E2 -10893} C_VEL
LIN {X 0,Y 402.863,Z 396.777,A -85,B 0,C 180,E1 -10894.001,E2 -10894.001} C_VEL
LIN {X 0,Y 402.893,Z 393.634,A -85,B 0,C 180,E1 -10895.505,E2 -10895.505} C_VEL
LIN {X 0,Y 403.004,Z 389.413,A -85,B 0,C 180,E1 -10897.012,E2 -10897.012} C_VEL
LIN {X 0,Y 403.301,Z 382.975,A -85,B 0,C 180,E1 -10898.77,E2 -10898.77} C_VEL
LIN {X 0,Y 403.686,Z 375.943,A -85,B 0,C 180,E1 -10900.279,E2 -10900.279} C_VEL
LIN {X 0,Y 404.331,Z 367.122,A -85,B 0,C 180,E1 -10901.785,E2 -10901.785} C_VEL
LIN {X 0,Y 404.965,Z 358.076,A -85,B 0,C 180,E1 -10903.039,E2 -10903.039} C_VEL
LIN {X 0,Y 405.593,Z 348.118,A -85,B 0,C 180,E1 -10904.167,E2 -10904.167} C_VEL
LIN {X 0,Y 406.384,Z 337.103,A -85,B 0,C 180,E1 -10905.163,E2 -10905.163} C_VEL
LIN {X 0,Y 407.153,Z 324.744,A -85,B 0,C 180,E1 -10906.032,E2 -10906.032} C_VEL
LIN {X 0,Y 407.808,Z 313.073,A -85,B 0,C 180,E1 -10906.649,E2 -10906.649} C_VEL
LIN {X 0,Y 408.423,Z 300.747,A -85,B 0,C 180,E1 -10907.106,E2 -10907.106} C_VEL
LIN {X 0,Y 408.675,Z 285.083,A -85,B 0,C 180,E1 -10907.45,E2 -10907.45} C_VEL
LIN {X 0,Y 409.361,Z 216.01,A -85,B 0,C 180,E1 -10908.677,E2 -10908.677} C_VEL
LIN {X 0,Y 405.407,Z 187.337,A -85,B 0,C 180,E1 -10909.395,E2 -10909.395} C_VEL
LIN {X 0,Y 406.631,Z 167.804,A -85,B 0,C 180,E1 -10913.153,E2 -10913.153} C_VEL
LIN {X 0,Y 407.125,Z 158.24,A -85,B 0,C 180,E1 -10915.02,E2 -10915.02} C_VEL
LIN {X 0,Y 404.749,Z 145.617,A -85,B 0,C 180,E1 -10917.679,E2 -10917.679} C_VEL
LIN {X 0,Y 404.226,Z 143.137,A -85,B 0,C 180,E1 -10918.244,E2 -10918.244} C_VEL
LIN {X 0,Y 404.141,Z 143.145,A -85,B 0,C 180,E1 -10921.558,E2 -10921.558} C_VEL
LIN {X 0,Y 404.186,Z 143.134,A -85,B 0,C 180,E1 -10925.016,E2 -10925.016} C_VEL
LIN {X 0,Y 404.158,Z 143.137,A -85,B 0,C 180,E1 -10928.756,E2 -10928.756} C_VEL
LIN {X 0,Y 404.124,Z 143.146,A -85,B 0,C 180,E1 -10931.6,E2 -10931.6} C_VEL
LIN {X 0,Y 404.146,Z 143.139,A -85,B 0,C 180,E1 -10934.522,E2 -10934.522} C_VEL
LIN {X 0,Y 404.137,Z 143.143,A -85,B 0,C 180,E1 -10937.295,E2 -10937.295} C_VEL
LIN {X 0,Y 404.169,Z 143.139,A -85,B 0,C 180,E1 -10939.955,E2 -10939.955} C_VEL
LIN {X 0,Y 404.136,Z 143.143,A -85,B 0,C 180,E1 -10943.125,E2 -10943.125} C_VEL
LIN {X 0,Y 404.145,Z 143.14,A -85,B 0,C 180,E1 -10946.187,E2 -10946.187} C_VEL
LIN {X 0,Y 404.146,Z 143.142,A -85,B 0,C 180,E1 -10949.715,E2 -10949.715} C_VEL
LIN {X 0,Y 404.196,Z 143.138,A -85,B 0,C 180,E1 -10953.123,E2 -10953.123} C_VEL
LIN {X 0,Y 404.175,Z 143.141,A -85,B 0,C 180,E1 -10955.334,E2 -10955.334} C_VEL
LIN {X 0,Y 404.138,Z 143.141,A -85,B 0,C 180,E1 -10958.58,E2 -10958.58} C_VEL
LIN {X 0,Y 404.205,Z 143.132,A -85,B 0,C 180,E1 -10961.761,E2 -10961.761} C_VEL
LIN {X 0,Y 404.206,Z 143.137,A -85,B 0,C 180,E1 -10964.882,E2 -10964.882} C_VEL
LIN {X 0,Y 404.256,Z 143.125,A -85,B 0,C 180,E1 -10967.958,E2 -10967.958} C_VEL
LIN {X 0,Y 404.266,Z 143.13,A -85,B 0,C 180,E1 -10970.998,E2 -10970.998} C_VEL
LIN {X 0,Y 404.394,Z 143.108,A -85,B 0,C 180,E1 -10974.014,E2 -10974.014} C_VEL
LIN {X 0,Y 404.481,Z 143.098,A -85,B 0,C 180,E1 -10978.008,E2 -10978.008} C_VEL
LIN {X 0,Y 404.609,Z 143.082,A -85,B 0,C 180,E1 -10980,E2 -10980} C_VEL
LIN {X 0,Y 404.421,Z 143.108,A -85,B 0,C 180,E1 -10982.988,E2 -10982.988} C_VEL
LIN {X 0,Y 404.399,Z 143.11,A -85,B 0,C 180,E1 -10986.987,E2 -10986.987} C_VEL
LIN {X 0,Y 404.257,Z 143.127,A -85,B 0,C 180,E1 -10990.012,E2 -10990.012} C_VEL
LIN {X 0,Y 404.266,Z 143.124,A -85,B 0,C 180,E1 -10993.211,E2 -10993.211} C_VEL
LIN {X 0,Y 404.215,Z 143.131,A -85,B 0,C 180,E1 -10997.007,E2 -10997.007} C_VEL
LIN {X 0,Y 404.163,Z 143.142,A -85,B 0,C 180,E1 -11000.351,E2 -11000.351} C_VEL
LIN {X 0,Y 404.162,Z 143.138,A -85,B 0,C 180,E1 -11003.575,E2 -11003.575} C_VEL
LIN {X 0,Y 404.182,Z 143.138,A -85,B 0,C 180,E1 -11005.766,E2 -11005.766} C_VEL
LIN {X 0,Y 404.194,Z 143.14,A -85,B 0,C 180,E1 -11008,E2 -11008} C_VEL
LIN {X 0,Y 404.138,Z 143.142,A -85,B 0,C 180,E1 -11011.558,E2 -11011.558} C_VEL
LIN {X 0,Y 404.183,Z 143.134,A -85,B 0,C 180,E1 -11015.016,E2 -11015.016} C_VEL
LIN {X 0,Y 404.156,Z 143.138,A -85,B 0,C 180,E1 -11018.757,E2 -11018.757} C_VEL
LIN {X 0,Y 404.122,Z 143.147,A -85,B 0,C 180,E1 -11021.6,E2 -11021.6} C_VEL
LIN {X 0,Y 404.144,Z 143.139,A -85,B 0,C 180,E1 -11024.522,E2 -11024.522} C_VEL
LIN {X 0,Y 404.135,Z 143.144,A -85,B 0,C 180,E1 -11027.296,E2 -11027.296} C_VEL
LIN {X 0,Y 404.168,Z 143.139,A -85,B 0,C 180,E1 -11029.955,E2 -11029.955} C_VEL
LIN {X 0,Y 404.134,Z 143.143,A -85,B 0,C 180,E1 -11033.125,E2 -11033.125} C_VEL
LIN {X 0,Y 404.143,Z 143.14,A -85,B 0,C 180,E1 -11036.188,E2 -11036.188} C_VEL
LIN {X 0,Y 404.145,Z 143.142,A -85,B 0,C 180,E1 -11039.715,E2 -11039.715} C_VEL
LIN {X 0,Y 404.195,Z 143.138,A -85,B 0,C 180,E1 -11043.123,E2 -11043.123} C_VEL
LIN {X 0,Y 404.174,Z 143.141,A -85,B 0,C 180,E1 -11045.334,E2 -11045.334} C_VEL
LIN {X 0,Y 404.138,Z 143.141,A -85,B 0,C 180,E1 -11048.581,E2 -11048.581} C_VEL
LIN {X 0,Y 404.204,Z 143.132,A -85,B 0,C 180,E1 -11051.762,E2 -11051.762} C_VEL
LIN {X 0,Y 404.206,Z 143.137,A -85,B 0,C 180,E1 -11054.882,E2 -11054.882} C_VEL
LIN {X 0,Y 404.256,Z 143.125,A -85,B 0,C 180,E1 -11057.959,E2 -11057.959} C_VEL
LIN {X 0,Y 404.266,Z 143.129,A -85,B 0,C 180,E1 -11060.999,E2 -11060.999} C_VEL
LIN {X 0,Y 404.394,Z 143.108,A -85,B 0,C 180,E1 -11064.015,E2 -11064.015} C_VEL
LIN {X 0,Y 404.474,Z 143.104,A -85,B 0,C 180,E1 -11068.258,E2 -11068.258} C_VEL
LIN {X 0,Y 404.462,Z 143.162,A -85,B 0,C 180,E1 -11068.382,E2 -11068.382} C_VEL
LIN {X 0,Y 405.822,Z 150.968,A -85,B 0,C 180,E1 -11070.273,E2 -11070.273} C_VEL
LIN {X 0,Y 405.962,Z 153.075,A -85,B 0,C 180,E1 -11070.741,E2 -11070.741} C_VEL
LIN {X 0,Y 409.894,Z 174.129,A -85,B 0,C 180,E1 -11071.298,E2 -11071.298} C_VEL
LIN {X 0,Y 408.709,Z 260.459,A -85,B 0,C 180,E1 -11072.849,E2 -11072.849} C_VEL
LIN {X 0,Y 408.341,Z 273.739,A -85,B 0,C 180,E1 -11073.291,E2 -11073.291} C_VEL
LIN {X 0,Y 408.312,Z 274.666,A -85,B 0,C 180,E1 -11073.329,E2 -11073.329} C_VEL
LIN {X 0,Y 407.645,Z 280.291,A -85,B 0,C 180,E1 -11073.563,E2 -11073.563} C_VEL
LIN {X 0,Y 404.457,Z 289.275,A -85,B 0,C 180,E1 -11073.957,E2 -11073.957} C_VEL
LIN {X 0,Y 401.084,Z 297.932,A -85,B 0,C 180,E1 -11074.459,E2 -11074.459} C_VEL
LIN {X 0,Y 400.138,Z 303.046,A -85,B 0,C 180,E1 -11074.86,E2 -11074.86} C_VEL
LIN {X 0,Y 399.393,Z 314.143,A -85,B 0,C 180,E1 -11075.934,E2 -11075.934} C_VEL
LIN {X 0,Y 398.676,Z 323.768,A -85,B 0,C 180,E1 -11077.088,E2 -11077.088} C_VEL
LIN {X 0,Y 397.892,Z 333.029,A -85,B 0,C 180,E1 -11078.456,E2 -11078.456} C_VEL
LIN {X 0,Y 397.293,Z 341.045,A -85,B 0,C 180,E1 -11079.932,E2 -11079.932} C_VEL
LIN {X 0,Y 396.772,Z 347.88,A -85,B 0,C 180,E1 -11081.494,E2 -11081.494} C_VEL
LIN {X 0,Y 396.382,Z 354.108,A -85,B 0,C 180,E1 -11083.326,E2 -11083.326} C_VEL
LIN {X 0,Y 396.073,Z 358.149,A -85,B 0,C 180,E1 -11084.91,E2 -11084.91} C_VEL
LIN {X 0,Y 395.865,Z 361.138,A -85,B 0,C 180,E1 -11086.527,E2 -11086.527} C_VEL
LIN {X 0,Y 395.763,Z 362.492,A -85,B 0,C 180,E1 -11087.571,E2 -11087.571} C_VEL
LIN {X 0,Y 395.734,Z 363.461,A -85,B 0,C 180,E1 -11088.643,E2 -11088.643} C_VEL
LIN {X 0,Y 395.722,Z 363.971,A -85,B 0,C 180,E1 -11089.733,E2 -11089.733} C_VEL
LIN {X 0,Y 395.716,Z 364.027,A -85,B 0,C 180,E1 -11090.806,E2 -11090.806} C_VEL
LIN {X 0,Y 395.806,Z 363.18,A -85,B 0,C 180,E1 -11092.584,E2 -11092.584} C_VEL
LIN {X 0,Y 395.999,Z 361.5,A -85,B 0,C 180,E1 -11094.092,E2 -11094.092} C_VEL
LIN {X 0,Y 396.304,Z 358.603,A -85,B 0,C 180,E1 -11095.752,E2 -11095.752} C_VEL
LIN {X 0,Y 396.663,Z 354.48,A -85,B 0,C 180,E1 -11097.43,E2 -11097.43} C_VEL
LIN {X 0,Y 397.201,Z 348.977,A -85,B 0,C 180,E1 -11099.116,E2 -11099.116} C_VEL
LIN {X 0,Y 397.921,Z 341.801,A -85,B 0,C 180,E1 -11100.81,E2 -11100.81} C_VEL
LIN {X 0,Y 398.732,Z 333.823,A -85,B 0,C 180,E1 -11102.312,E2 -11102.312} C_VEL
LIN {X 0,Y 399.633,Z 325.111,A -85,B 0,C 180,E1 -11103.64,E2 -11103.64} C_VEL
LIN {X 0,Y 400.457,Z 315.875,A -85,B 0,C 180,E1 -11104.787,E2 -11104.787} C_VEL
LIN {X 0,Y 401.439,Z 304.648,A -85,B 0,C 180,E1 -11105.908,E2 -11105.908} C_VEL
LIN {X 0,Y 402.399,Z 292.587,A -85,B 0,C 180,E1 -11106.849,E2 -11106.849} C_VEL
LIN {X 0,Y 403.004,Z 281.157,A -85,B 0,C 180,E1 -11107.53,E2 -11107.53} C_VEL
LIN {X 0,Y 403.533,Z 268.618,A -85,B 0,C 180,E1 -11108.066,E2 -11108.066} C_VEL
LIN {X 0,Y 403.865,Z 255.5,A -85,B 0,C 180,E1 -11108.422,E2 -11108.422} C_VEL
LIN {X 0,Y 405.104,Z 174.569,A -85,B 0,C 180,E1 -11109.906,E2 -11109.906} C_VEL
LIN {X 0,Y 402.029,Z 161.369,A -85,B 0,C 180,E1 -11110.353,E2 -11110.353} C_VEL
LIN {X 0,Y 399.188,Z 153.822,A -85,B 0,C 180,E1 -11110.699,E2 -11110.699} C_VEL
LIN {X 0,Y 397.094,Z 144.025,A -85,B 0,C 180,E1 -11113.293,E2 -11113.293} C_VEL
LIN {X 0,Y 397.096,Z 144.028,A -85,B 0,C 180,E1 -11116.522,E2 -11116.522} C_VEL
LIN {X 0,Y 397.086,Z 144.017,A -85,B 0,C 180,E1 -11120.42,E2 -11120.42} C_VEL
LIN {X 0,Y 397.097,Z 144.015,A -85,B 0,C 180,E1 -11123.005,E2 -11123.005} C_VEL
LIN {X 0,Y 397.111,Z 144.02,A -85,B 0,C 180,E1 -11126.727,E2 -11126.727} C_VEL
LIN {X 0,Y 397.115,Z 144.021,A -85,B 0,C 180,E1 -11130.295,E2 -11130.295} C_VEL
LIN {X 0,Y 397.072,Z 144.023,A -85,B 0,C 180,E1 -11133.737,E2 -11133.737} C_VEL
LIN {X 0,Y 397.099,Z 144.015,A -85,B 0,C 180,E1 -11137.085,E2 -11137.085} C_VEL
LIN {X 0,Y 397.094,Z 144.02,A -85,B 0,C 180,E1 -11140.35,E2 -11140.35} C_VEL
LIN {X 0,Y 397.115,Z 144.017,A -85,B 0,C 180,E1 -11143.551,E2 -11143.551} C_VEL
LIN {X 0,Y 397.192,Z 144.009,A -85,B 0,C 180,E1 -11146.702,E2 -11146.702} C_VEL
LIN {X 0,Y 397.203,Z 144,A -85,B 0,C 180,E1 -11149.809,E2 -11149.809} C_VEL
LIN {X 0,Y 397.294,Z 143.988,A -85,B 0,C 180,E1 -11152.887,E2 -11152.887} C_VEL
LIN {X 0,Y 397.227,Z 144,A -85,B 0,C 180,E1 -11154.925,E2 -11154.925} C_VEL
LIN {X 0,Y 397.438,Z 143.971,A -85,B 0,C 180,E1 -11157.973,E2 -11157.973} C_VEL
LIN {X 0,Y 397.319,Z 143.99,A -85,B 0,C 180,E1 -11161.014,E2 -11161.014} C_VEL
LIN {X 0,Y 397.322,Z 143.982,A -85,B 0,C 180,E1 -11163.042,E2 -11163.042} C_VEL
LIN {X 0,Y 397.329,Z 143.989,A -85,B 0,C 180,E1 -11166.092,E2 -11166.092} C_VEL
LIN {X 0,Y 397.232,Z 143.999,A -85,B 0,C 180,E1 -11169.163,E2 -11169.163} C_VEL
LIN {X 0,Y 397.22,Z 143.997,A -85,B 0,C 180,E1 -11172.258,E2 -11172.258} C_VEL
LIN {X 0,Y 397.177,Z 144.014,A -85,B 0,C 180,E1 -11175.392,E2 -11175.392} C_VEL
LIN {X 0,Y 397.159,Z 144.005,A -85,B 0,C 180,E1 -11178.574,E2 -11178.574} C_VEL
LIN {X 0,Y 397.099,Z 144.011,A -85,B 0,C 180,E1 -11181.819,E2 -11181.819} C_VEL
LIN {X 0,Y 397.11,Z 144.018,A -85,B 0,C 180,E1 -11185.135,E2 -11185.135} C_VEL
LIN {X 0,Y 397.074,Z 144.023,A -85,B 0,C 180,E1 -11188.548,E2 -11188.548} C_VEL
LIN {X 0,Y 397.083,Z 144.02,A -85,B 0,C 180,E1 -11191.836,E2 -11191.836} C_VEL
LIN {X 0,Y 397.127,Z 144.013,A -85,B 0,C 180,E1 -11194.493,E2 -11194.493} C_VEL
LIN {X 0,Y 397.096,Z 144.018,A -85,B 0,C 180,E1 -11198.276,E2 -11198.276} C_VEL
LIN {X 0,Y 397.061,Z 144.026,A -85,B 0,C 180,E1 -11201.978,E2 -11201.978} C_VEL
LIN {X 0,Y 397.089,Z 144.022,A -85,B 0,C 180,E1 -11205.069,E2 -11205.069} C_VEL
LIN {X 0,Y 397.065,Z 144.027,A -85,B 0,C 180,E1 -11208.022,E2 -11208.022} C_VEL
LIN {X 0,Y 397.126,Z 144.017,A -85,B 0,C 180,E1 -11211.14,E2 -11211.14} C_VEL
LIN {X 0,Y 397.121,Z 144.017,A -85,B 0,C 180,E1 -11214.497,E2 -11214.497} C_VEL
LIN {X 0,Y 397.081,Z 144.022,A -85,B 0,C 180,E1 -11217.928,E2 -11217.928} C_VEL
LIN {X 0,Y 397.127,Z 144.064,A -85,B 0,C 180,E1 -11220.296,E2 -11220.296} C_VEL
LIN {X 0,Y 399.573,Z 154.601,A -85,B 0,C 180,E1 -11222.786,E2 -11222.786} C_VEL
LIN {X 0,Y 401.074,Z 162.558,A -85,B 0,C 180,E1 -11224.576,E2 -11224.576} C_VEL
LIN {X 0,Y 400.807,Z 167.304,A -85,B 0,C 180,E1 -11225.548,E2 -11225.548} C_VEL
LIN {X 0,Y 399.304,Z 186.329,A -85,B 0,C 180,E1 -11229.365,E2 -11229.365} C_VEL
LIN {X 0,Y 403.581,Z 210.904,A -85,B 0,C 180,E1 -11230.113,E2 -11230.113} C_VEL
LIN {X 0,Y 404.464,Z 219.242,A -85,B 0,C 180,E1 -11230.326,E2 -11230.326} C_VEL
LIN {X 0,Y 403.337,Z 295.673,A -85,B 0,C 180,E1 -11231.754,E2 -11231.754} C_VEL
LIN {X 0,Y 402.676,Z 308.672,A -85,B 0,C 180,E1 -11232.183,E2 -11232.183} C_VEL
LIN {X 0,Y 401.938,Z 320.697,A -85,B 0,C 180,E1 -11232.773,E2 -11232.773} C_VEL
LIN {X 0,Y 400.943,Z 332.926,A -85,B 0,C 180,E1 -11233.581,E2 -11233.581} C_VEL
LIN {X 0,Y 399.894,Z 344.506,A -85,B 0,C 180,E1 -11234.584,E2 -11234.584} C_VEL
LIN {X 0,Y 398.954,Z 354.953,A -85,B 0,C 180,E1 -11235.722,E2 -11235.722} C_VEL
LIN {X 0,Y 398.122,Z 364.389,A -85,B 0,C 180,E1 -11236.993,E2 -11236.993} C_VEL
LIN {X 0,Y 397.214,Z 373.508,A -85,B 0,C 180,E1 -11238.518,E2 -11238.518} C_VEL
LIN {X 0,Y 396.589,Z 380.881,A -85,B 0,C 180,E1 -11240.05,E2 -11240.05} C_VEL
LIN {X 0,Y 396.157,Z 387.673,A -85,B 0,C 180,E1 -11241.841,E2 -11241.841} C_VEL
LIN {X 0,Y 395.876,Z 392.299,A -85,B 0,C 180,E1 -11243.425,E2 -11243.425} C_VEL
LIN {X 0,Y 395.828,Z 395.604,A -85,B 0,C 180,E1 -11244.907,E2 -11244.907} C_VEL
LIN {X 0,Y 395.779,Z 397.316,A -85,B 0,C 180,E1 -11245.927,E2 -11245.927} C_VEL
LIN {X 0,Y 395.858,Z 399.546,A -85,B 0,C 180,E1 -11247.965,E2 -11247.965} C_VEL
LIN {X 0,Y 395.834,Z 400.028,A -85,B 0,C 180,E1 -11248.982,E2 -11248.982} C_VEL
LIN {X 0,Y 395.825,Z 400.103,A -85,B 0,C 180,E1 -11250,E2 -11250} C_VEL
LIN {X 0,Y 395.879,Z 399.089,A -85,B 0,C 180,E1 -11252.035,E2 -11252.035} C_VEL
LIN {X 0,Y 395.791,Z 397.948,A -85,B 0,C 180,E1 -11253.053,E2 -11253.053} C_VEL
LIN {X 0,Y 395.785,Z 396.373,A -85,B 0,C 180,E1 -11254.073,E2 -11254.073} C_VEL
LIN {X 0,Y 395.795,Z 392.822,A -85,B 0,C 180,E1 -11255.757,E2 -11255.757} C_VEL
LIN {X 0,Y 396.032,Z 387.292,A -85,B 0,C 180,E1 -11257.648,E2 -11257.648} C_VEL
LIN {X 0,Y 396.373,Z 380.257,A -85,B 0,C 180,E1 -11259.44,E2 -11259.44} C_VEL
LIN {X 0,Y 396.835,Z 372.635,A -85,B 0,C 180,E1 -11260.975,E2 -11260.975} C_VEL
LIN {X 0,Y 397.47,Z 364.852,A -85,B 0,C 180,E1 -11262.25,E2 -11262.25} C_VEL
LIN {X 0,Y 398.191,Z 354.899,A -85,B 0,C 180,E1 -11263.577,E2 -11263.577} C_VEL
LIN {X 0,Y 398.896,Z 344.762,A -85,B 0,C 180,E1 -11264.671,E2 -11264.671} C_VEL
LIN {X 0,Y 399.679,Z 332.999,A -85,B 0,C 180,E1 -11265.685,E2 -11265.685} C_VEL
LIN {X 0,Y 400.52,Z 320.447,A -85,B 0,C 180,E1 -11266.502,E2 -11266.502} C_VEL
LIN {X 0,Y 401.206,Z 307.214,A -85,B 0,C 180,E1 -11267.128,E2 -11267.128} C_VEL
LIN {X 0,Y 401.663,Z 295.306,A -85,B 0,C 180,E1 -11267.501,E2 -11267.501} C_VEL
LIN {X 0,Y 402.578,Z 217.136,A -85,B 0,C 180,E1 -11268.93,E2 -11268.93} C_VEL
LIN {X 0,Y 398.445,Z 187.073,A -85,B 0,C 180,E1 -11269.681,E2 -11269.681} C_VEL
LIN {X 0,Y 399.668,Z 168.563,A -85,B 0,C 180,E1 -11273.307,E2 -11273.307} C_VEL
LIN {X 0,Y 400.184,Z 160.38,A -85,B 0,C 180,E1 -11274.928,E2 -11274.928} C_VEL
LIN {X 0,Y 398.79,Z 152.007,A -85,B 0,C 180,E1 -11276.704,E2 -11276.704} C_VEL
LIN {X 0,Y 397.193,Z 144.013,A -85,B 0,C 180,E1 -11278.445,E2 -11278.445} C_VEL
LIN {X 0,Y 397.08,Z 144.025,A -85,B 0,C 180,E1 -11282.071,E2 -11282.071} C_VEL
LIN {X 0,Y 397.12,Z 144.016,A -85,B 0,C 180,E1 -11285.503,E2 -11285.503} C_VEL
LIN {X 0,Y 397.133,Z 144.012,A -85,B 0,C 180,E1 -11288.861,E2 -11288.861} C_VEL
LIN {X 0,Y 397.07,Z 144.022,A -85,B 0,C 180,E1 -11292.267,E2 -11292.267} C_VEL
LIN {X 0,Y 397.087,Z 144.019,A -85,B 0,C 180,E1 -11295.068,E2 -11295.068} C_VEL
LIN {X 0,Y 397.067,Z 144.024,A -85,B 0,C 180,E1 -11298.021,E2 -11298.021} C_VEL
LIN {X 0,Y 397.127,Z 144.016,A -85,B 0,C 180,E1 -11301.139,E2 -11301.139} C_VEL
LIN {X 0,Y 397.119,Z 144.014,A -85,B 0,C 180,E1 -11304.497,E2 -11304.497} C_VEL
LIN {X 0,Y 397.078,Z 144.021,A -85,B 0,C 180,E1 -11307.928,E2 -11307.928} C_VEL
LIN {X 0,Y 397.123,Z 144.019,A -85,B 0,C 180,E1 -11311.456,E2 -11311.456} C_VEL
LIN {X 0,Y 397.153,Z 144.01,A -85,B 0,C 180,E1 -11314.487,E2 -11314.487} C_VEL
LIN {X 0,Y 397.096,Z 144.017,A -85,B 0,C 180,E1 -11318.181,E2 -11318.181} C_VEL
LIN {X 0,Y 397.158,Z 144.013,A -85,B 0,C 180,E1 -11321.426,E2 -11321.426} C_VEL
LIN {X 0,Y 397.179,Z 144.009,A -85,B 0,C 180,E1 -11324.608,E2 -11324.608} C_VEL
LIN {X 0,Y 397.219,Z 144.002,A -85,B 0,C 180,E1 -11327.742,E2 -11327.742} C_VEL
LIN {X 0,Y 397.236,Z 144.006,A -85,B 0,C 180,E1 -11330.838,E2 -11330.838} C_VEL
LIN {X 0,Y 397.345,Z 143.986,A -85,B 0,C 180,E1 -11333.908,E2 -11333.908} C_VEL
LIN {X 0,Y 397.449,Z 143.974,A -85,B 0,C 180,E1 -11337.973,E2 -11337.973} C_VEL
LIN {X 0,Y 397.579,Z 143.958,A -85,B 0,C 180,E1 -11340,E2 -11340} C_VEL
LIN {X 0,Y 397.379,Z 143.984,A -85,B 0,C 180,E1 -11343.041,E2 -11343.041} C_VEL
LIN {X 0,Y 397.344,Z 143.986,A -85,B 0,C 180,E1 -11346.581,E2 -11346.581} C_VEL
LIN {X 0,Y 397.252,Z 143.998,A -85,B 0,C 180,E1 -11349.162,E2 -11349.162} C_VEL
LIN {X 0,Y 397.218,Z 144.007,A -85,B 0,C 180,E1 -11352.258,E2 -11352.258} C_VEL
LIN {X 0,Y 397.178,Z 144.007,A -85,B 0,C 180,E1 -11355.392,E2 -11355.392} C_VEL
LIN {X 0,Y 397.16,Z 144.013,A -85,B 0,C 180,E1 -11358.573,E2 -11358.573} C_VEL
LIN {X 0,Y 397.095,Z 144.02,A -85,B 0,C 180,E1 -11361.818,E2 -11361.818} C_VEL
LIN {X 0,Y 397.151,Z 144.011,A -85,B 0,C 180,E1 -11365.512,E2 -11365.512} C_VEL
LIN {X 0,Y 397.121,Z 144.016,A -85,B 0,C 180,E1 -11368.544,E2 -11368.544} C_VEL
LIN {X 0,Y 397.078,Z 144.025,A -85,B 0,C 180,E1 -11372.071,E2 -11372.071} C_VEL
LIN {X 0,Y 397.118,Z 144.017,A -85,B 0,C 180,E1 -11375.503,E2 -11375.503} C_VEL
LIN {X 0,Y 397.131,Z 144.013,A -85,B 0,C 180,E1 -11378.862,E2 -11378.862} C_VEL
LIN {X 0,Y 397.068,Z 144.022,A -85,B 0,C 180,E1 -11382.267,E2 -11382.267} C_VEL
LIN {X 0,Y 397.085,Z 144.02,A -85,B 0,C 180,E1 -11385.069,E2 -11385.069} C_VEL
LIN {X 0,Y 397.065,Z 144.023,A -85,B 0,C 180,E1 -11388.021,E2 -11388.021} C_VEL
LIN {X 0,Y 397.125,Z 144.016,A -85,B 0,C 180,E1 -11391.139,E2 -11391.139} C_VEL
LIN {X 0,Y 397.117,Z 144.014,A -85,B 0,C 180,E1 -11394.497,E2 -11394.497} C_VEL
LIN {X 0,Y 397.077,Z 144.021,A -85,B 0,C 180,E1 -11397.928,E2 -11397.928} C_VEL
LIN {X 0,Y 397.122,Z 144.019,A -85,B 0,C 180,E1 -11401.457,E2 -11401.457} C_VEL
LIN {X 0,Y 397.152,Z 144.011,A -85,B 0,C 180,E1 -11404.488,E2 -11404.488} C_VEL
LIN {X 0,Y 397.095,Z 144.017,A -85,B 0,C 180,E1 -11408.182,E2 -11408.182} C_VEL
LIN {X 0,Y 397.158,Z 144.012,A -85,B 0,C 180,E1 -11411.427,E2 -11411.427} C_VEL
LIN {X 0,Y 397.179,Z 144.01,A -85,B 0,C 180,E1 -11414.608,E2 -11414.608} C_VEL
LIN {X 0,Y 397.219,Z 144.002,A -85,B 0,C 180,E1 -11417.742,E2 -11417.742} C_VEL
LIN {X 0,Y 397.235,Z 144.007,A -85,B 0,C 180,E1 -11420.838,E2 -11420.838} C_VEL
LIN {X 0,Y 397.346,Z 143.986,A -85,B 0,C 180,E1 -11423.908,E2 -11423.908} C_VEL
LIN {X 0,Y 397.446,Z 144.08,A -85,B 0,C 180,E1 -11428.195,E2 -11428.195} C_VEL
LIN {X 0,Y 398.958,Z 153.176,A -85,B 0,C 180,E1 -11430.426,E2 -11430.426} C_VEL
LIN {X 0,Y 402.996,Z 173.775,A -85,B 0,C 180,E1 -11430.999,E2 -11430.999} C_VEL
LIN {X 0,Y 401.855,Z 260.993,A -85,B 0,C 180,E1 -11432.6,E2 -11432.6} C_VEL
LIN {X 0,Y 401.461,Z 274.347,A -85,B 0,C 180,E1 -11433.056,E2 -11433.056} C_VEL
LIN {X 0,Y 401.006,Z 286.6,A -85,B 0,C 180,E1 -11433.674,E2 -11433.674} C_VEL
LIN {X 0,Y 400.449,Z 297.439,A -85,B 0,C 180,E1 -11434.404,E2 -11434.404} C_VEL
LIN {X 0,Y 400.138,Z 303.046,A -85,B 0,C 180,E1 -11434.86,E2 -11434.86} C_VEL
LIN {X 0,Y 399.219,Z 308.102,A -85,B 0,C 180,E1 -11435.297,E2 -11435.297} C_VEL
LIN {X 0,Y 395.847,Z 316.006,A -85,B 0,C 180,E1 -11436.019,E2 -11436.019} C_VEL
LIN {X 0,Y 392.412,Z 323.409,A -85,B 0,C 180,E1 -11436.831,E2 -11436.831} C_VEL
LIN {X 0,Y 391.394,Z 327.647,A -85,B 0,C 180,E1 -11437.404,E2 -11437.404} C_VEL
LIN {X 0,Y 390.672,Z 336.304,A -85,B 0,C 180,E1 -11438.808,E2 -11438.808} C_VEL
LIN {X 0,Y 390.038,Z 344.074,A -85,B 0,C 180,E1 -11440.381,E2 -11440.381} C_VEL
LIN {X 0,Y 389.576,Z 350.351,A -85,B 0,C 180,E1 -11441.974,E2 -11441.974} C_VEL
LIN {X 0,Y 389.239,Z 355.324,A -85,B 0,C 180,E1 -11443.576,E2 -11443.576} C_VEL
LIN {X 0,Y 388.938,Z 359.147,A -85,B 0,C 180,E1 -11445.19,E2 -11445.19} C_VEL
LIN {X 0,Y 388.758,Z 361.89,A -85,B 0,C 180,E1 -11446.813,E2 -11446.813} C_VEL
LIN {X 0,Y 388.662,Z 363.177,A -85,B 0,C 180,E1 -11447.903,E2 -11447.903} C_VEL
LIN {X 0,Y 388.622,Z 364.315,A -85,B 0,C 180,E1 -11449.883,E2 -11449.883} C_VEL
LIN {X 0,Y 388.652,Z 364.307,A -85,B 0,C 180,E1 -11451.202,E2 -11451.202} C_VEL
LIN {X 0,Y 388.743,Z 363.431,A -85,B 0,C 180,E1 -11452.778,E2 -11452.778} C_VEL
LIN {X 0,Y 388.995,Z 361.356,A -85,B 0,C 180,E1 -11454.554,E2 -11454.554} C_VEL
LIN {X 0,Y 389.315,Z 358.216,A -85,B 0,C 180,E1 -11456.25,E2 -11456.25} C_VEL
LIN {X 0,Y 389.76,Z 353.802,A -85,B 0,C 180,E1 -11457.958,E2 -11457.958} C_VEL
LIN {X 0,Y 390.354,Z 347.969,A -85,B 0,C 180,E1 -11459.678,E2 -11459.678} C_VEL
LIN {X 0,Y 391.193,Z 340.501,A -85,B 0,C 180,E1 -11461.4,E2 -11461.4} C_VEL
LIN {X 0,Y 392.026,Z 332.633,A -85,B 0,C 180,E1 -11462.841,E2 -11462.841} C_VEL
LIN {X 0,Y 393.02,Z 322.871,A -85,B 0,C 180,E1 -11464.283,E2 -11464.283} C_VEL
LIN {X 0,Y 393.997,Z 313.241,A -85,B 0,C 180,E1 -11465.431,E2 -11465.431} C_VEL
LIN {X 0,Y 395.023,Z 301.82,A -85,B 0,C 180,E1 -11466.518,E2 -11466.518} C_VEL
LIN {X 0,Y 395.925,Z 289.228,A -85,B 0,C 180,E1 -11467.443,E2 -11467.443} C_VEL
LIN {X 0,Y 396.59,Z 277.416,A -85,B 0,C 180,E1 -11468.091,E2 -11468.091} C_VEL
LIN {X 0,Y 397.06,Z 264.573,A -85,B 0,C 180,E1 -11468.579,E2 -11468.579} C_VEL
LIN {X 0,Y 397.435,Z 246.777,A -85,B 0,C 180,E1 -11468.964,E2 -11468.964} C_VEL
LIN {X 0,Y 398.654,Z 176.007,A -85,B 0,C 180,E1 -11470.278,E2 -11470.278} C_VEL
LIN {X 0,Y 395.763,Z 163.659,A -85,B 0,C 180,E1 -11470.708,E2 -11470.708} C_VEL
LIN {X 0,Y 392.039,Z 154.19,A -85,B 0,C 180,E1 -11471.156,E2 -11471.156} C_VEL
LIN {X 0,Y 390.051,Z 144.903,A -85,B 0,C 180,E1 -11473.654,E2 -11473.654} C_VEL
LIN {X 0,Y 390.051,Z 144.903,A -85,B 0,C 180,E1 -11476.789,E2 -11476.789} C_VEL
LIN {X 0,Y 390.009,Z 144.902,A -85,B 0,C 180,E1 -11479.555,E2 -11479.555} C_VEL
LIN {X 0,Y 390.04,Z 144.901,A -85,B 0,C 180,E1 -11482.45,E2 -11482.45} C_VEL
LIN {X 0,Y 390.061,Z 144.896,A -85,B 0,C 180,E1 -11486.045,E2 -11486.045} C_VEL
LIN {X 0,Y 390.042,Z 144.901,A -85,B 0,C 180,E1 -11489.871,E2 -11489.871} C_VEL
LIN {X 0,Y 390.027,Z 144.902,A -85,B 0,C 180,E1 -11493.226,E2 -11493.226} C_VEL
LIN {X 0,Y 390.058,Z 144.896,A -85,B 0,C 180,E1 -11496.768,E2 -11496.768} C_VEL
LIN {X 0,Y 390.068,Z 144.897,A -85,B 0,C 180,E1 -11499.981,E2 -11499.981} C_VEL
LIN {X 0,Y 390.08,Z 144.893,A -85,B 0,C 180,E1 -11503.246,E2 -11503.246} C_VEL
LIN {X 0,Y 390.133,Z 144.89,A -85,B 0,C 180,E1 -11506.601,E2 -11506.601} C_VEL
LIN {X 0,Y 390.155,Z 144.876,A -85,B 0,C 180,E1 -11509.623,E2 -11509.623} C_VEL
LIN {X 0,Y 390.247,Z 144.866,A -85,B 0,C 180,E1 -11512.758,E2 -11512.758} C_VEL
LIN {X 0,Y 390.198,Z 144.876,A -85,B 0,C 180,E1 -11514.833,E2 -11514.833} C_VEL
LIN {X 0,Y 390.404,Z 144.847,A -85,B 0,C 180,E1 -11517.937,E2 -11517.937} C_VEL
LIN {X 0,Y 390.408,Z 144.846,A -85,B 0,C 180,E1 -11522.063,E2 -11522.063} C_VEL
LIN {X 0,Y 390.283,Z 144.866,A -85,B 0,C 180,E1 -11526.203,E2 -11526.203} C_VEL
LIN {X 0,Y 390.191,Z 144.877,A -85,B 0,C 180,E1 -11529.329,E2 -11529.329} C_VEL
LIN {X 0,Y 390.172,Z 144.874,A -85,B 0,C 180,E1 -11532.483,E2 -11532.483} C_VEL
LIN {X 0,Y 390.138,Z 144.887,A -85,B 0,C 180,E1 -11535.677,E2 -11535.677} C_VEL
LIN {X 0,Y 390.104,Z 144.886,A -85,B 0,C 180,E1 -11538.922,E2 -11538.922} C_VEL
LIN {X 0,Y 390.041,Z 144.889,A -85,B 0,C 180,E1 -11542.234,E2 -11542.234} C_VEL
LIN {X 0,Y 390.052,Z 144.892,A -85,B 0,C 180,E1 -11545.722,E2 -11545.722} C_VEL
LIN {X 0,Y 390.032,Z 144.9,A -85,B 0,C 180,E1 -11549.112,E2 -11549.112} C_VEL
LIN {X 0,Y 390.045,Z 144.902,A -85,B 0,C 180,E1 -11552.722,E2 -11552.722} C_VEL
LIN {X 0,Y 390.058,Z 144.896,A -85,B 0,C 180,E1 -11555.825,E2 -11555.825} C_VEL
LIN {X 0,Y 390.04,Z 144.9,A -85,B 0,C 180,E1 -11559.213,E2 -11559.213} C_VEL
LIN {X 0,Y 390.039,Z 144.904,A -85,B 0,C 180,E1 -11562.373,E2 -11562.373} C_VEL
LIN {X 0,Y 390.046,Z 144.899,A -85,B 0,C 180,E1 -11565.354,E2 -11565.354} C_VEL
LIN {X 0,Y 390.03,Z 144.903,A -85,B 0,C 180,E1 -11568.186,E2 -11568.186} C_VEL
LIN {X 0,Y 390.085,Z 144.895,A -85,B 0,C 180,E1 -11570.907,E2 -11570.907} C_VEL
LIN {X 0,Y 390.087,Z 144.89,A -85,B 0,C 180,E1 -11574.793,E2 -11574.793} C_VEL
LIN {X 0,Y 390.027,Z 144.904,A -85,B 0,C 180,E1 -11578.496,E2 -11578.496} C_VEL
LIN {X 0,Y 390.066,Z 144.972,A -85,B 0,C 180,E1 -11579.9,E2 -11579.9} C_VEL
LIN {X 0,Y 392.405,Z 154.636,A -85,B 0,C 180,E1 -11582.247,E2 -11582.247} C_VEL
LIN {X 0,Y 394.162,Z 163.861,A -85,B 0,C 180,E1 -11584.381,E2 -11584.381} C_VEL
LIN {X 0,Y 394.056,Z 167.645,A -85,B 0,C 180,E1 -11585.181,E2 -11585.181} C_VEL
LIN {X 0,Y 392.444,Z 185.962,A -85,B 0,C 180,E1 -11588.92,E2 -11588.92} C_VEL
LIN {X 0,Y 396.032,Z 205.368,A -85,B 0,C 180,E1 -11589.545,E2 -11589.545} C_VEL
LIN {X 0,Y 397.911,Z 218.551,A -85,B 0,C 180,E1 -11589.921,E2 -11589.921} C_VEL
LIN {X 0,Y 396.734,Z 295.19,A -85,B 0,C 180,E1 -11591.376,E2 -11591.376} C_VEL
LIN {X 0,Y 396.017,Z 308.906,A -85,B 0,C 180,E1 -11591.84,E2 -11591.84} C_VEL
LIN {X 0,Y 395.265,Z 320.223,A -85,B 0,C 180,E1 -11592.406,E2 -11592.406} C_VEL
LIN {X 0,Y 394.346,Z 331.644,A -85,B 0,C 180,E1 -11593.165,E2 -11593.165} C_VEL
LIN {X 0,Y 393.216,Z 343.403,A -85,B 0,C 180,E1 -11594.183,E2 -11594.183} C_VEL
LIN {X 0,Y 392.161,Z 353.96,A -85,B 0,C 180,E1 -11595.337,E2 -11595.337} C_VEL
LIN {X 0,Y 391.317,Z 362.613,A -85,B 0,C 180,E1 -11596.498,E2 -11596.498} C_VEL
LIN {X 0,Y 390.593,Z 370.61,A -85,B 0,C 180,E1 -11597.794,E2 -11597.794} C_VEL
LIN {X 0,Y 389.759,Z 378.49,A -85,B 0,C 180,E1 -11599.349,E2 -11599.349} C_VEL
LIN {X 0,Y 389.213,Z 385.725,A -85,B 0,C 180,E1 -11601.171,E2 -11601.171} C_VEL
LIN {X 0,Y 388.903,Z 390.581,A -85,B 0,C 180,E1 -11602.732,E2 -11602.732} C_VEL
LIN {X 0,Y 388.752,Z 393.477,A -85,B 0,C 180,E1 -11603.888,E2 -11603.888} C_VEL
LIN {X 0,Y 388.703,Z 397.053,A -85,B 0,C 180,E1 -11605.852,E2 -11605.852} C_VEL
LIN {X 0,Y 388.756,Z 399.251,A -85,B 0,C 180,E1 -11607.928,E2 -11607.928} C_VEL
LIN {X 0,Y 388.763,Z 399.711,A -85,B 0,C 180,E1 -11608.964,E2 -11608.964} C_VEL
LIN {X 0,Y 388.753,Z 399.772,A -85,B 0,C 180,E1 -11610,E2 -11610} C_VEL
LIN {X 0,Y 388.764,Z 399.446,A -85,B 0,C 180,E1 -11611.036,E2 -11611.036} C_VEL
LIN {X 0,Y 388.791,Z 398.728,A -85,B 0,C 180,E1 -11612.072,E2 -11612.072} C_VEL
LIN {X 0,Y 388.694,Z 397.558,A -85,B 0,C 180,E1 -11613.109,E2 -11613.109} C_VEL
LIN {X 0,Y 388.715,Z 395.034,A -85,B 0,C 180,E1 -11614.667,E2 -11614.667} C_VEL
LIN {X 0,Y 388.72,Z 391.477,A -85,B 0,C 180,E1 -11616.227,E2 -11616.227} C_VEL
LIN {X 0,Y 388.965,Z 386.804,A -85,B 0,C 180,E1 -11617.788,E2 -11617.788} C_VEL
LIN {X 0,Y 389.319,Z 379.728,A -85,B 0,C 180,E1 -11619.612,E2 -11619.612} C_VEL
LIN {X 0,Y 389.83,Z 372.062,A -85,B 0,C 180,E1 -11621.175,E2 -11621.175} C_VEL
LIN {X 0,Y 390.467,Z 364.216,A -85,B 0,C 180,E1 -11622.473,E2 -11622.473} C_VEL
LIN {X 0,Y 391.204,Z 353.694,A -85,B 0,C 180,E1 -11623.883,E2 -11623.883} C_VEL
LIN {X 0,Y 392.057,Z 342.655,A -85,B 0,C 180,E1 -11625.066,E2 -11625.066} C_VEL
LIN {X 0,Y 392.829,Z 332.054,A -85,B 0,C 180,E1 -11625.966,E2 -11625.966} C_VEL
LIN {X 0,Y 393.633,Z 319.284,A -85,B 0,C 180,E1 -11626.799,E2 -11626.799} C_VEL
LIN {X 0,Y 394.359,Z 306.536,A -85,B 0,C 180,E1 -11627.401,E2 -11627.401} C_VEL
LIN {X 0,Y 394.822,Z 294.332,A -85,B 0,C 180,E1 -11627.781,E2 -11627.781} C_VEL
LIN {X 0,Y 395.717,Z 217.37,A -85,B 0,C 180,E1 -11629.212,E2 -11629.212} C_VEL
LIN {X 0,Y 391.489,Z 186.803,A -85,B 0,C 180,E1 -11629.977,E2 -11629.977} C_VEL
LIN {X 0,Y 392.808,Z 168.022,A -85,B 0,C 180,E1 -11633.726,E2 -11633.726} C_VEL
LIN {X 0,Y 393.201,Z 161.143,A -85,B 0,C 180,E1 -11635.119,E2 -11635.119} C_VEL
LIN {X 0,Y 390.882,Z 148.516,A -85,B 0,C 180,E1 -11637.87,E2 -11637.87} C_VEL
LIN {X 0,Y 390.147,Z 144.889,A -85,B 0,C 180,E1 -11638.702,E2 -11638.702} C_VEL
LIN {X 0,Y 390.044,Z 144.896,A -85,B 0,C 180,E1 -11642.721,E2 -11642.721} C_VEL
LIN {X 0,Y 390.057,Z 144.9,A -85,B 0,C 180,E1 -11645.825,E2 -11645.825} C_VEL
LIN {X 0,Y 390.072,Z 144.893,A -85,B 0,C 180,E1 -11649.218,E2 -11649.218} C_VEL
LIN {X 0,Y 390.044,Z 144.897,A -85,B 0,C 180,E1 -11652.374,E2 -11652.374} C_VEL
LIN {X 0,Y 390.045,Z 144.899,A -85,B 0,C 180,E1 -11655.354,E2 -11655.354} C_VEL
LIN {X 0,Y 390.032,Z 144.899,A -85,B 0,C 180,E1 -11658.186,E2 -11658.186} C_VEL
LIN {X 0,Y 390.088,Z 144.891,A -85,B 0,C 180,E1 -11660.907,E2 -11660.907} C_VEL
LIN {X 0,Y 390.085,Z 144.891,A -85,B 0,C 180,E1 -11664.793,E2 -11664.793} C_VEL
LIN {X 0,Y 390.023,Z 144.898,A -85,B 0,C 180,E1 -11668.495,E2 -11668.495} C_VEL
LIN {X 0,Y 390.118,Z 144.887,A -85,B 0,C 180,E1 -11672.07,E2 -11672.07} C_VEL
LIN {X 0,Y 390.078,Z 144.895,A -85,B 0,C 180,E1 -11675.519,E2 -11675.519} C_VEL
LIN {X 0,Y 390.055,Z 144.898,A -85,B 0,C 180,E1 -11678.878,E2 -11678.878} C_VEL
LIN {X 0,Y 390.111,Z 144.887,A -85,B 0,C 180,E1 -11682.166,E2 -11682.166} C_VEL
LIN {X 0,Y 390.144,Z 144.886,A -85,B 0,C 180,E1 -11685.392,E2 -11685.392} C_VEL
LIN {X 0,Y 390.147,Z 144.886,A -85,B 0,C 180,E1 -11688.571,E2 -11688.571} C_VEL
LIN {X 0,Y 390.258,Z 144.869,A -85,B 0,C 180,E1 -11692.083,E2 -11692.083} C_VEL
LIN {X 0,Y 390.218,Z 144.881,A -85,B 0,C 180,E1 -11694.833,E2 -11694.833} C_VEL
LIN {X 0,Y 390.418,Z 144.849,A -85,B 0,C 180,E1 -11697.937,E2 -11697.937} C_VEL
LIN {X 0,Y 390.548,Z 144.834,A -85,B 0,C 180,E1 -11700,E2 -11700} C_VEL
LIN {X 0,Y 390.313,Z 144.864,A -85,B 0,C 180,E1 -11703.096,E2 -11703.096} C_VEL
LIN {X 0,Y 390.301,Z 144.864,A -85,B 0,C 180,E1 -11706.575,E2 -11706.575} C_VEL
LIN {X 0,Y 390.204,Z 144.876,A -85,B 0,C 180,E1 -11709.329,E2 -11709.329} C_VEL
LIN {X 0,Y 390.194,Z 144.877,A -85,B 0,C 180,E1 -11713.438,E2 -11713.438} C_VEL
LIN {X 0,Y 390.148,Z 144.883,A -85,B 0,C 180,E1 -11717.308,E2 -11717.308} C_VEL
LIN {X 0,Y 390.086,Z 144.894,A -85,B 0,C 180,E1 -11720.47,E2 -11720.47} C_VEL
LIN {X 0,Y 390.072,Z 144.892,A -85,B 0,C 180,E1 -11723.352,E2 -11723.352} C_VEL
LIN {X 0,Y 390.112,Z 144.888,A -85,B 0,C 180,E1 -11726.768,E2 -11726.768} C_VEL
LIN {X 0,Y 390.038,Z 144.9,A -85,B 0,C 180,E1 -11730.3,E2 -11730.3} C_VEL
LIN {X 0,Y 390.067,Z 144.898,A -85,B 0,C 180,E1 -11734.025,E2 -11734.025} C_VEL
LIN {X 0,Y 390.043,Z 144.899,A -85,B 0,C 180,E1 -11737.551,E2 -11737.551} C_VEL
LIN {X 0,Y 390.056,Z 144.894,A -85,B 0,C 180,E1 -11740.821,E2 -11740.821} C_VEL
LIN {X 0,Y 390.053,Z 144.899,A -85,B 0,C 180,E1 -11743.886,E2 -11743.886} C_VEL
LIN {X 0,Y 390.056,Z 144.894,A -85,B 0,C 180,E1 -11746.79,E2 -11746.79} C_VEL
LIN {X 0,Y 390.055,Z 144.901,A -85,B 0,C 180,E1 -11749.561,E2 -11749.561} C_VEL
LIN {X 0,Y 390.041,Z 144.896,A -85,B 0,C 180,E1 -11752.45,E2 -11752.45} C_VEL
LIN {X 0,Y 390.067,Z 144.894,A -85,B 0,C 180,E1 -11755.976,E2 -11755.976} C_VEL
LIN {X 0,Y 390.046,Z 144.897,A -85,B 0,C 180,E1 -11759.869,E2 -11759.869} C_VEL
LIN {X 0,Y 390.113,Z 144.894,A -85,B 0,C 180,E1 -11763.232,E2 -11763.232} C_VEL
LIN {X 0,Y 390.076,Z 144.894,A -85,B 0,C 180,E1 -11766.761,E2 -11766.761} C_VEL
LIN {X 0,Y 390.103,Z 144.888,A -85,B 0,C 180,E1 -11769.983,E2 -11769.983} C_VEL
LIN {X 0,Y 390.138,Z 144.888,A -85,B 0,C 180,E1 -11773.248,E2 -11773.248} C_VEL
LIN {X 0,Y 390.194,Z 144.88,A -85,B 0,C 180,E1 -11776.562,E2 -11776.562} C_VEL
LIN {X 0,Y 390.167,Z 144.881,A -85,B 0,C 180,E1 -11779.623,E2 -11779.623} C_VEL
LIN {X 0,Y 390.268,Z 144.874,A -85,B 0,C 180,E1 -11782.758,E2 -11782.758} C_VEL
LIN {X 0,Y 390.218,Z 144.88,A -85,B 0,C 180,E1 -11784.834,E2 -11784.834} C_VEL
LIN {X 0,Y 390.419,Z 145.002,A -85,B 0,C 180,E1 -11788.001,E2 -11788.001} C_VEL
LIN {X 0,Y 391.922,Z 153.633,A -85,B 0,C 180,E1 -11790.131,E2 -11790.131} C_VEL
LIN {X 0,Y 395.877,Z 172.743,A -85,B 0,C 180,E1 -11790.67,E2 -11790.67} C_VEL
LIN {X 0,Y 396.26,Z 177.243,A -85,B 0,C 180,E1 -11790.772,E2 -11790.772} C_VEL
LIN {X 0,Y 395.011,Z 260.866,A -85,B 0,C 180,E1 -11792.323,E2 -11792.323} C_VEL
LIN {X 0,Y 394.603,Z 274.66,A -85,B 0,C 180,E1 -11792.799,E2 -11792.799} C_VEL
LIN {X 0,Y 394.16,Z 286.643,A -85,B 0,C 180,E1 -11793.414,E2 -11793.414} C_VEL
LIN {X 0,Y 393.518,Z 298.425,A -85,B 0,C 180,E1 -11794.225,E2 -11794.225} C_VEL
LIN {X 0,Y 392.772,Z 310.038,A -85,B 0,C 180,E1 -11795.262,E2 -11795.262} C_VEL
LIN {X 0,Y 391.983,Z 320.517,A -85,B 0,C 180,E1 -11796.434,E2 -11796.434} C_VEL
LIN {X 0,Y 391.394,Z 327.647,A -85,B 0,C 180,E1 -11797.404,E2 -11797.404} C_VEL
LIN {X 0,Y 390.402,Z 331.774,A -85,B 0,C 180,E1 -11798.008,E2 -11798.008} C_VEL
LIN {X 0,Y 387.042,Z 338.133,A -85,B 0,C 180,E1 -11799.019,E2 -11799.019} C_VEL
LIN {X 0,Y 383.729,Z 343.838,A -85,B 0,C 180,E1 -11800.121,E2 -11800.121} C_VEL
LIN {X 0,Y 382.821,Z 346.937,A -85,B 0,C 180,E1 -11800.861,E2 -11800.861} C_VEL
LIN {X 0,Y 382.323,Z 353.482,A -85,B 0,C 180,E1 -11802.744,E2 -11802.744} C_VEL
LIN {X 0,Y 381.993,Z 357.831,A -85,B 0,C 180,E1 -11804.382,E2 -11804.382} C_VEL
LIN {X 0,Y 381.74,Z 361.07,A -85,B 0,C 180,E1 -11806.031,E2 -11806.031} C_VEL
LIN {X 0,Y 381.631,Z 362.667,A -85,B 0,C 180,E1 -11807.137,E2 -11807.137} C_VEL
LIN {X 0,Y 381.572,Z 363.772,A -85,B 0,C 180,E1 -11808.247,E2 -11808.247} C_VEL
LIN {X 0,Y 381.566,Z 364.661,A -85,B 0,C 180,E1 -11810.056,E2 -11810.056} C_VEL
LIN {X 0,Y 381.564,Z 364.51,A -85,B 0,C 180,E1 -11811.616,E2 -11811.616} C_VEL
LIN {X 0,Y 381.7,Z 363.68,A -85,B 0,C 180,E1 -11812.984,E2 -11812.984} C_VEL
LIN {X 0,Y 381.803,Z 362.757,A -85,B 0,C 180,E1 -11813.889,E2 -11813.889} C_VEL
LIN {X 0,Y 382.145,Z 360,A -85,B 0,C 180,E1 -11815.69,E2 -11815.69} C_VEL
LIN {X 0,Y 382.522,Z 356.363,A -85,B 0,C 180,E1 -11817.343,E2 -11817.343} C_VEL
LIN {X 0,Y 383.085,Z 351.227,A -85,B 0,C 180,E1 -11819.089,E2 -11819.089} C_VEL
LIN {X 0,Y 383.851,Z 344.57,A -85,B 0,C 180,E1 -11820.841,E2 -11820.841} C_VEL
LIN {X 0,Y 384.653,Z 337.767,A -85,B 0,C 180,E1 -11822.272,E2 -11822.272} C_VEL
LIN {X 0,Y 385.655,Z 328.987,A -85,B 0,C 180,E1 -11823.767,E2 -11823.767} C_VEL
LIN {X 0,Y 386.674,Z 319.09,A -85,B 0,C 180,E1 -11825.125,E2 -11825.125} C_VEL
LIN {X 0,Y 387.726,Z 308.85,A -85,B 0,C 180,E1 -11826.254,E2 -11826.254} C_VEL
LIN {X 0,Y 388.713,Z 298.243,A -85,B 0,C 180,E1 -11827.189,E2 -11827.189} C_VEL
LIN {X 0,Y 389.488,Z 286.331,A -85,B 0,C 180,E1 -11828.007,E2 -11828.007} C_VEL
LIN {X 0,Y 390.181,Z 273.166,A -85,B 0,C 180,E1 -11828.667,E2 -11828.667} C_VEL
LIN {X 0,Y 390.58,Z 260.119,A -85,B 0,C 180,E1 -11829.096,E2 -11829.096} C_VEL
LIN {X 0,Y 392.1,Z 176.748,A -85,B 0,C 180,E1 -11830.684,E2 -11830.684} C_VEL
LIN {X 0,Y 389.495,Z 165.839,A -85,B 0,C 180,E1 -11831.078,E2 -11831.078} C_VEL
LIN {X 0,Y 384.931,Z 154.518,A -85,B 0,C 180,E1 -11831.645,E2 -11831.645} C_VEL
LIN {X 0,Y 383.01,Z 145.781,A -85,B 0,C 180,E1 -11834.079,E2 -11834.079} C_VEL
LIN {X 0,Y 383.011,Z 145.777,A -85,B 0,C 180,E1 -11837.24,E2 -11837.24} C_VEL
LIN {X 0,Y 382.985,Z 145.774,A -85,B 0,C 180,E1 -11840.419,E2 -11840.419} C_VEL
LIN {X 0,Y 383.015,Z 145.768,A -85,B 0,C 180,E1 -11844.044,E2 -11844.044} C_VEL
LIN {X 0,Y 382.983,Z 145.78,A -85,B 0,C 180,E1 -11847.579,E2 -11847.579} C_VEL
LIN {X 0,Y 382.975,Z 145.783,A -85,B 0,C 180,E1 -11850.299,E2 -11850.299} C_VEL
LIN {X 0,Y 383.003,Z 145.777,A -85,B 0,C 180,E1 -11854.045,E2 -11854.045} C_VEL
LIN {X 0,Y 382.983,Z 145.772,A -85,B 0,C 180,E1 -11857.334,E2 -11857.334} C_VEL
LIN {X 0,Y 383.011,Z 145.771,A -85,B 0,C 180,E1 -11860.714,E2 -11860.714} C_VEL
LIN {X 0,Y 383.002,Z 145.776,A -85,B 0,C 180,E1 -11864.024,E2 -11864.024} C_VEL
LIN {X 0,Y 383.109,Z 145.761,A -85,B 0,C 180,E1 -11867.283,E2 -11867.283} C_VEL
LIN {X 0,Y 383.136,Z 145.76,A -85,B 0,C 180,E1 -11870.498,E2 -11870.498} C_VEL
LIN {X 0,Y 383.201,Z 145.745,A -85,B 0,C 180,E1 -11872.624,E2 -11872.624} C_VEL
LIN {X 0,Y 383.17,Z 145.752,A -85,B 0,C 180,E1 -11874.738,E2 -11874.738} C_VEL
LIN {X 0,Y 383.369,Z 145.723,A -85,B 0,C 180,E1 -11877.899,E2 -11877.899} C_VEL
LIN {X 0,Y 383.374,Z 145.722,A -85,B 0,C 180,E1 -11882.101,E2 -11882.101} C_VEL
LIN {X 0,Y 383.24,Z 145.743,A -85,B 0,C 180,E1 -11886.317,E2 -11886.317} C_VEL
LIN {X 0,Y 383.142,Z 145.757,A -85,B 0,C 180,E1 -11889.503,E2 -11889.503} C_VEL
LIN {X 0,Y 383.128,Z 145.754,A -85,B 0,C 180,E1 -11893.536,E2 -11893.536} C_VEL
LIN {X 0,Y 383.096,Z 145.76,A -85,B 0,C 180,E1 -11897.069,E2 -11897.069} C_VEL
LIN {X 0,Y 383.031,Z 145.771,A -85,B 0,C 180,E1 -11900.647,E2 -11900.647} C_VEL
LIN {X 0,Y 383.021,Z 145.772,A -85,B 0,C 180,E1 -11903.808,E2 -11903.808} C_VEL
LIN {X 0,Y 382.989,Z 145.775,A -85,B 0,C 180,E1 -11907.307,E2 -11907.307} C_VEL
LIN {X 0,Y 382.984,Z 145.775,A -85,B 0,C 180,E1 -11910.919,E2 -11910.919} C_VEL
LIN {X 0,Y 383.02,Z 145.771,A -85,B 0,C 180,E1 -11914.668,E2 -11914.668} C_VEL
LIN {X 0,Y 382.996,Z 145.773,A -85,B 0,C 180,E1 -11917.903,E2 -11917.903} C_VEL
LIN {X 0,Y 382.965,Z 145.782,A -85,B 0,C 180,E1 -11921.35,E2 -11921.35} C_VEL
LIN {X 0,Y 382.997,Z 145.78,A -85,B 0,C 180,E1 -11924.303,E2 -11924.303} C_VEL
LIN {X 0,Y 383.013,Z 145.777,A -85,B 0,C 180,E1 -11927.24,E2 -11927.24} C_VEL
LIN {X 0,Y 383.012,Z 145.778,A -85,B 0,C 180,E1 -11930.415,E2 -11930.415} C_VEL
LIN {X 0,Y 383.027,Z 145.776,A -85,B 0,C 180,E1 -11934.044,E2 -11934.044} C_VEL
LIN {X 0,Y 382.989,Z 145.777,A -85,B 0,C 180,E1 -11937.578,E2 -11937.578} C_VEL
LIN {X 0,Y 382.984,Z 145.78,A -85,B 0,C 180,E1 -11939.462,E2 -11939.462} C_VEL
LIN {X 0,Y 385.471,Z 155.986,A -85,B 0,C 180,E1 -11941.999,E2 -11941.999} C_VEL
LIN {X 0,Y 387.266,Z 165.212,A -85,B 0,C 180,E1 -11944.18,E2 -11944.18} C_VEL
LIN {X 0,Y 387.166,Z 169.304,A -85,B 0,C 180,E1 -11945.065,E2 -11945.065} C_VEL
LIN {X 0,Y 385.627,Z 185.631,A -85,B 0,C 180,E1 -11948.468,E2 -11948.468} C_VEL
LIN {X 0,Y 389.432,Z 205.689,A -85,B 0,C 180,E1 -11949.133,E2 -11949.133} C_VEL
LIN {X 0,Y 391.382,Z 220.283,A -85,B 0,C 180,E1 -11949.551,E2 -11949.551} C_VEL
LIN {X 0,Y 390.142,Z 294.728,A -85,B 0,C 180,E1 -11950.985,E2 -11950.985} C_VEL
LIN {X 0,Y 389.409,Z 308.388,A -85,B 0,C 180,E1 -11951.452,E2 -11951.452} C_VEL
LIN {X 0,Y 388.547,Z 320.871,A -85,B 0,C 180,E1 -11952.092,E2 -11952.092} C_VEL
LIN {X 0,Y 387.578,Z 332.036,A -85,B 0,C 180,E1 -11952.862,E2 -11952.862} C_VEL
LIN {X 0,Y 386.404,Z 343.635,A -85,B 0,C 180,E1 -11953.896,E2 -11953.896} C_VEL
LIN {X 0,Y 385.293,Z 354.096,A -85,B 0,C 180,E1 -11955.069,E2 -11955.069} C_VEL
LIN {X 0,Y 384.394,Z 362.672,A -85,B 0,C 180,E1 -11956.25,E2 -11956.25} C_VEL
LIN {X 0,Y 383.643,Z 370.603,A -85,B 0,C 180,E1 -11957.57,E2 -11957.57} C_VEL
LIN {X 0,Y 382.75,Z 378.39,A -85,B 0,C 180,E1 -11959.152,E2 -11959.152} C_VEL
LIN {X 0,Y 382.171,Z 385.569,A -85,B 0,C 180,E1 -11961.007,E2 -11961.007} C_VEL
LIN {X 0,Y 381.838,Z 390.381,A -85,B 0,C 180,E1 -11962.597,E2 -11962.597} C_VEL
LIN {X 0,Y 381.67,Z 393.512,A -85,B 0,C 180,E1 -11963.906,E2 -11963.906} C_VEL
LIN {X 0,Y 381.626,Z 396.79,A -85,B 0,C 180,E1 -11965.775,E2 -11965.775} C_VEL
LIN {X 0,Y 381.654,Z 398.952,A -85,B 0,C 180,E1 -11967.889,E2 -11967.889} C_VEL
LIN {X 0,Y 381.694,Z 399.393,A -85,B 0,C 180,E1 -11968.945,E2 -11968.945} C_VEL
LIN {X 0,Y 381.682,Z 399.441,A -85,B 0,C 180,E1 -11970,E2 -11970} C_VEL
LIN {X 0,Y 381.695,Z 399.101,A -85,B 0,C 180,E1 -11971.055,E2 -11971.055} C_VEL
LIN {X 0,Y 381.69,Z 398.362,A -85,B 0,C 180,E1 -11972.11,E2 -11972.11} C_VEL
LIN {X 0,Y 381.6,Z 397.168,A -85,B 0,C 180,E1 -11973.167,E2 -11973.167} C_VEL
LIN {X 0,Y 381.632,Z 394.614,A -85,B 0,C 180,E1 -11974.753,E2 -11974.753} C_VEL
LIN {X 0,Y 381.652,Z 391.025,A -85,B 0,C 180,E1 -11976.343,E2 -11976.343} C_VEL
LIN {X 0,Y 381.883,Z 386.314,A -85,B 0,C 180,E1 -11977.933,E2 -11977.933} C_VEL
LIN {X 0,Y 382.266,Z 379.199,A -85,B 0,C 180,E1 -11979.791,E2 -11979.791} C_VEL
LIN {X 0,Y 382.842,Z 371.482,A -85,B 0,C 180,E1 -11981.381,E2 -11981.381} C_VEL
LIN {X 0,Y 383.455,Z 363.567,A -85,B 0,C 180,E1 -11982.705,E2 -11982.705} C_VEL
LIN {X 0,Y 384.181,Z 354.009,A -85,B 0,C 180,E1 -11984.012,E2 -11984.012} C_VEL
LIN {X 0,Y 385.046,Z 343.142,A -85,B 0,C 180,E1 -11985.211,E2 -11985.211} C_VEL
LIN {X 0,Y 385.846,Z 332.754,A -85,B 0,C 180,E1 -11986.127,E2 -11986.127} C_VEL
LIN {X 0,Y 386.673,Z 320.333,A -85,B 0,C 180,E1 -11986.974,E2 -11986.974} C_VEL
LIN {X 0,Y 387.452,Z 307.278,A -85,B 0,C 180,E1 -11987.619,E2 -11987.619} C_VEL
LIN {X 0,Y 387.969,Z 294.546,A -85,B 0,C 180,E1 -11988.038,E2 -11988.038} C_VEL
LIN {X 0,Y 388.925,Z 218.459,A -85,B 0,C 180,E1 -11989.476,E2 -11989.476} C_VEL
LIN {X 0,Y 384.569,Z 186.37,A -85,B 0,C 180,E1 -11990.317,E2 -11990.317} C_VEL
LIN {X 0,Y 385.924,Z 168.066,A -85,B 0,C 180,E1 -11994.043,E2 -11994.043} C_VEL
LIN {X 0,Y 386.206,Z 161.876,A -85,B 0,C 180,E1 -11995.318,E2 -11995.318} C_VEL
LIN {X 0,Y 383.506,Z 147.79,A -85,B 0,C 180,E1 -11998.455,E2 -11998.455} C_VEL
LIN {X 0,Y 383.079,Z 145.769,A -85,B 0,C 180,E1 -11998.939,E2 -11998.939} C_VEL
LIN {X 0,Y 382.988,Z 145.777,A -85,B 0,C 180,E1 -12002.422,E2 -12002.422} C_VEL
LIN {X 0,Y 383.026,Z 145.776,A -85,B 0,C 180,E1 -12005.955,E2 -12005.955} C_VEL
LIN {X 0,Y 383.017,Z 145.775,A -85,B 0,C 180,E1 -12009.586,E2 -12009.586} C_VEL
LIN {X 0,Y 383.006,Z 145.772,A -85,B 0,C 180,E1 -12012.778,E2 -12012.778} C_VEL
LIN {X 0,Y 382.998,Z 145.779,A -85,B 0,C 180,E1 -12015.789,E2 -12015.789} C_VEL
LIN {X 0,Y 382.988,Z 145.775,A -85,B 0,C 180,E1 -12018.796,E2 -12018.796} C_VEL
LIN {X 0,Y 382.998,Z 145.775,A -85,B 0,C 180,E1 -12022.096,E2 -12022.096} C_VEL
LIN {X 0,Y 383.018,Z 145.776,A -85,B 0,C 180,E1 -12025.332,E2 -12025.332} C_VEL
LIN {X 0,Y 382.983,Z 145.779,A -85,B 0,C 180,E1 -12029.081,E2 -12029.081} C_VEL
LIN {X 0,Y 383.057,Z 145.767,A -85,B 0,C 180,E1 -12032.698,E2 -12032.698} C_VEL
LIN {X 0,Y 383.051,Z 145.771,A -85,B 0,C 180,E1 -12035.039,E2 -12035.039} C_VEL
LIN {X 0,Y 382.992,Z 145.775,A -85,B 0,C 180,E1 -12038.469,E2 -12038.469} C_VEL
LIN {X 0,Y 383.053,Z 145.767,A -85,B 0,C 180,E1 -12041.826,E2 -12041.826} C_VEL
LIN {X 0,Y 383.11,Z 145.765,A -85,B 0,C 180,E1 -12045.118,E2 -12045.118} C_VEL
LIN {X 0,Y 383.097,Z 145.762,A -85,B 0,C 180,E1 -12048.358,E2 -12048.358} C_VEL
LIN {X 0,Y 383.22,Z 145.746,A -85,B 0,C 180,E1 -12052.022,E2 -12052.022} C_VEL
LIN {X 0,Y 383.189,Z 145.756,A -85,B 0,C 180,E1 -12054.738,E2 -12054.738} C_VEL
LIN {X 0,Y 383.386,Z 145.725,A -85,B 0,C 180,E1 -12057.899,E2 -12057.899} C_VEL
LIN {X 0,Y 383.517,Z 145.709,A -85,B 0,C 180,E1 -12060,E2 -12060} C_VEL
LIN {X 0,Y 383.249,Z 145.744,A -85,B 0,C 180,E1 -12063.153,E2 -12063.153} C_VEL
LIN {X 0,Y 383.262,Z 145.742,A -85,B 0,C 180,E1 -12066.566,E2 -12066.566} C_VEL
LIN {X 0,Y 383.151,Z 145.754,A -85,B 0,C 180,E1 -12069.502,E2 -12069.502} C_VEL
LIN {X 0,Y 383.125,Z 145.758,A -85,B 0,C 180,E1 -12073.536,E2 -12073.536} C_VEL
LIN {X 0,Y 383.094,Z 145.762,A -85,B 0,C 180,E1 -12077.454,E2 -12077.454} C_VEL
LIN {X 0,Y 383.028,Z 145.772,A -85,B 0,C 180,E1 -12080.647,E2 -12080.647} C_VEL
LIN {X 0,Y 383.024,Z 145.773,A -85,B 0,C 180,E1 -12083.808,E2 -12083.808} C_VEL
LIN {X 0,Y 383.079,Z 145.77,A -85,B 0,C 180,E1 -12086.123,E2 -12086.123} C_VEL
LIN {X 0,Y 382.991,Z 145.778,A -85,B 0,C 180,E1 -12089.7,E2 -12089.7} C_VEL
LIN {X 0,Y 383.011,Z 145.773,A -85,B 0,C 180,E1 -12093.4,E2 -12093.4} C_VEL
LIN {X 0,Y 383.031,Z 145.773,A -85,B 0,C 180,E1 -12096.165,E2 -12096.165} C_VEL
LIN {X 0,Y 383.008,Z 145.777,A -85,B 0,C 180,E1 -12099.958,E2 -12099.958} C_VEL
LIN {X 0,Y 383.004,Z 145.773,A -85,B 0,C 180,E1 -12102.779,E2 -12102.779} C_VEL
LIN {X 0,Y 382.996,Z 145.779,A -85,B 0,C 180,E1 -12105.789,E2 -12105.789} C_VEL
LIN {X 0,Y 382.986,Z 145.775,A -85,B 0,C 180,E1 -12108.796,E2 -12108.796} C_VEL
LIN {X 0,Y 382.997,Z 145.775,A -85,B 0,C 180,E1 -12112.097,E2 -12112.097} C_VEL
LIN {X 0,Y 383.016,Z 145.777,A -85,B 0,C 180,E1 -12115.332,E2 -12115.332} C_VEL
LIN {X 0,Y 382.982,Z 145.779,A -85,B 0,C 180,E1 -12119.082,E2 -12119.082} C_VEL
LIN {X 0,Y 383.056,Z 145.768,A -85,B 0,C 180,E1 -12122.698,E2 -12122.698} C_VEL
LIN {X 0,Y 383.05,Z 145.772,A -85,B 0,C 180,E1 -12125.04,E2 -12125.04} C_VEL
LIN {X 0,Y 382.992,Z 145.775,A -85,B 0,C 180,E1 -12128.469,E2 -12128.469} C_VEL
LIN {X 0,Y 383.052,Z 145.767,A -85,B 0,C 180,E1 -12131.826,E2 -12131.826} C_VEL
LIN {X 0,Y 383.11,Z 145.765,A -85,B 0,C 180,E1 -12135.118,E2 -12135.118} C_VEL
LIN {X 0,Y 383.097,Z 145.763,A -85,B 0,C 180,E1 -12138.358,E2 -12138.358} C_VEL
LIN {X 0,Y 383.22,Z 145.746,A -85,B 0,C 180,E1 -12142.022,E2 -12142.022} C_VEL
LIN {X 0,Y 383.189,Z 145.756,A -85,B 0,C 180,E1 -12144.739,E2 -12144.739} C_VEL
LIN {X 0,Y 383.37,Z 145.816,A -85,B 0,C 180,E1 -12147.768,E2 -12147.768} C_VEL
LIN {X 0,Y 384.81,Z 153.827,A -85,B 0,C 180,E1 -12149.804,E2 -12149.804} C_VEL
LIN {X 0,Y 387.112,Z 163.538,A -85,B 0,C 180,E1 -12150.103,E2 -12150.103} C_VEL
LIN {X 0,Y 389.472,Z 176.642,A -85,B 0,C 180,E1 -12150.465,E2 -12150.465} C_VEL
LIN {X 0,Y 388.154,Z 261.677,A -85,B 0,C 180,E1 -12152.075,E2 -12152.075} C_VEL
LIN {X 0,Y 387.764,Z 274.499,A -85,B 0,C 180,E1 -12152.525,E2 -12152.525} C_VEL
LIN {X 0,Y 387.278,Z 287.137,A -85,B 0,C 180,E1 -12153.18,E2 -12153.18} C_VEL
LIN {X 0,Y 386.585,Z 299.297,A -85,B 0,C 180,E1 -12154.04,E2 -12154.04} C_VEL
LIN {X 0,Y 385.811,Z 310.825,A -85,B 0,C 180,E1 -12155.095,E2 -12155.095} C_VEL
LIN {X 0,Y 384.981,Z 321.231,A -85,B 0,C 180,E1 -12156.289,E2 -12156.289} C_VEL
LIN {X 0,Y 384.165,Z 330.56,A -85,B 0,C 180,E1 -12157.622,E2 -12157.622} C_VEL
LIN {X 0,Y 383.426,Z 339.477,A -85,B 0,C 180,E1 -12159.203,E2 -12159.203} C_VEL
LIN {X 0,Y 382.821,Z 346.937,A -85,B 0,C 180,E1 -12160.861,E2 -12160.861} C_VEL
LIN {X 0,Y 381.94,Z 349.877,A -85,B 0,C 180,E1 -12161.625,E2 -12161.625} C_VEL
LIN {X 0,Y 377.344,Z 355.72,A -85,B 0,C 180,E1 -12163.398,E2 -12163.398} C_VEL
LIN {X 0,Y 375.189,Z 358.479,A -85,B 0,C 180,E1 -12164.483,E2 -12164.483} C_VEL
LIN {X 0,Y 374.784,Z 359.67,A -85,B 0,C 180,E1 -12165.054,E2 -12165.054} C_VEL
LIN {X 0,Y 374.561,Z 362.644,A -85,B 0,C 180,E1 -12166.878,E2 -12166.878} C_VEL
LIN {X 0,Y 374.452,Z 364.35,A -85,B 0,C 180,E1 -12168.607,E2 -12168.607} C_VEL
LIN {X 0,Y 374.485,Z 365.004,A -85,B 0,C 180,E1 -12170.223,E2 -12170.223} C_VEL
LIN {X 0,Y 374.498,Z 364.693,A -85,B 0,C 180,E1 -12172.045,E2 -12172.045} C_VEL
LIN {X 0,Y 374.631,Z 363.923,A -85,B 0,C 180,E1 -12173.201,E2 -12173.201} C_VEL
LIN {X 0,Y 374.791,Z 362.64,A -85,B 0,C 180,E1 -12174.365,E2 -12174.365} C_VEL
LIN {X 0,Y 375.112,Z 360.183,A -85,B 0,C 180,E1 -12175.932,E2 -12175.932} C_VEL
LIN {X 0,Y 375.623,Z 355.787,A -85,B 0,C 180,E1 -12177.889,E2 -12177.889} C_VEL
LIN {X 0,Y 376.254,Z 350.396,A -85,B 0,C 180,E1 -12179.669,E2 -12179.669} C_VEL
LIN {X 0,Y 377.146,Z 343.375,A -85,B 0,C 180,E1 -12181.451,E2 -12181.451} C_VEL
LIN {X 0,Y 378.022,Z 335.968,A -85,B 0,C 180,E1 -12182.955,E2 -12182.955} C_VEL
LIN {X 0,Y 379.12,Z 327.001,A -85,B 0,C 180,E1 -12184.43,E2 -12184.43} C_VEL
LIN {X 0,Y 380.144,Z 317.72,A -85,B 0,C 180,E1 -12185.671,E2 -12185.671} C_VEL
LIN {X 0,Y 381.247,Z 307.118,A -85,B 0,C 180,E1 -12186.807,E2 -12186.807} C_VEL
LIN {X 0,Y 382.266,Z 295.866,A -85,B 0,C 180,E1 -12187.762,E2 -12187.762} C_VEL
LIN {X 0,Y 383.055,Z 284.282,A -85,B 0,C 180,E1 -12188.528,E2 -12188.528} C_VEL
LIN {X 0,Y 383.69,Z 271.756,A -85,B 0,C 180,E1 -12189.13,E2 -12189.13} C_VEL
LIN {X 0,Y 384.077,Z 258.95,A -85,B 0,C 180,E1 -12189.527,E2 -12189.527} C_VEL
LIN {X 0,Y 385.604,Z 177.898,A -85,B 0,C 180,E1 -12191.095,E2 -12191.095} C_VEL
LIN {X 0,Y 383.469,Z 168.716,A -85,B 0,C 180,E1 -12191.435,E2 -12191.435} C_VEL
LIN {X 0,Y 377.795,Z 154.889,A -85,B 0,C 180,E1 -12192.156,E2 -12192.156} C_VEL
LIN {X 0,Y 375.944,Z 146.66,A -85,B 0,C 180,E1 -12194.524,E2 -12194.524} C_VEL
LIN {X 0,Y 375.925,Z 146.659,A -85,B 0,C 180,E1 -12197.699,E2 -12197.699} C_VEL
LIN {X 0,Y 375.934,Z 146.652,A -85,B 0,C 180,E1 -12200.534,E2 -12200.534} C_VEL
LIN {X 0,Y 375.958,Z 146.645,A -85,B 0,C 180,E1 -12203.497,E2 -12203.497} C_VEL
LIN {X 0,Y 375.957,Z 146.653,A -85,B 0,C 180,E1 -12205.889,E2 -12205.889} C_VEL
LIN {X 0,Y 375.96,Z 146.655,A -85,B 0,C 180,E1 -12209.687,E2 -12209.687} C_VEL
LIN {X 0,Y 375.916,Z 146.659,A -85,B 0,C 180,E1 -12212.135,E2 -12212.135} C_VEL
LIN {X 0,Y 375.935,Z 146.656,A -85,B 0,C 180,E1 -12214.534,E2 -12214.534} C_VEL
LIN {X 0,Y 375.969,Z 146.649,A -85,B 0,C 180,E1 -12216.887,E2 -12216.887} C_VEL
LIN {X 0,Y 375.959,Z 146.653,A -85,B 0,C 180,E1 -12220.337,E2 -12220.337} C_VEL
LIN {X 0,Y 375.954,Z 146.653,A -85,B 0,C 180,E1 -12223.716,E2 -12223.716} C_VEL
LIN {X 0,Y 376.076,Z 146.638,A -85,B 0,C 180,E1 -12227.041,E2 -12227.041} C_VEL
LIN {X 0,Y 376.107,Z 146.634,A -85,B 0,C 180,E1 -12230.318,E2 -12230.318} C_VEL
LIN {X 0,Y 376.194,Z 146.616,A -85,B 0,C 180,E1 -12233.564,E2 -12233.564} C_VEL
LIN {X 0,Y 376.333,Z 146.599,A -85,B 0,C 180,E1 -12237.86,E2 -12237.86} C_VEL
LIN {X 0,Y 376.338,Z 146.597,A -85,B 0,C 180,E1 -12242.141,E2 -12242.141} C_VEL
LIN {X 0,Y 376.199,Z 146.619,A -85,B 0,C 180,E1 -12246.436,E2 -12246.436} C_VEL
LIN {X 0,Y 376.113,Z 146.635,A -85,B 0,C 180,E1 -12249.682,E2 -12249.682} C_VEL
LIN {X 0,Y 376.092,Z 146.632,A -85,B 0,C 180,E1 -12253.658,E2 -12253.658} C_VEL
LIN {X 0,Y 376.034,Z 146.637,A -85,B 0,C 180,E1 -12257.4,E2 -12257.4} C_VEL
LIN {X 0,Y 375.981,Z 146.651,A -85,B 0,C 180,E1 -12260.832,E2 -12260.832} C_VEL
LIN {X 0,Y 375.977,Z 146.649,A -85,B 0,C 180,E1 -12264.283,E2 -12264.283} C_VEL
LIN {X 0,Y 375.931,Z 146.654,A -85,B 0,C 180,E1 -12267.864,E2 -12267.864} C_VEL
LIN {X 0,Y 375.959,Z 146.652,A -85,B 0,C 180,E1 -12271.562,E2 -12271.562} C_VEL
LIN {X 0,Y 375.959,Z 146.653,A -85,B 0,C 180,E1 -12275.416,E2 -12275.416} C_VEL
LIN {X 0,Y 375.939,Z 146.654,A -85,B 0,C 180,E1 -12278.263,E2 -12278.263} C_VEL
LIN {X 0,Y 375.921,Z 146.659,A -85,B 0,C 180,E1 -12281.598,E2 -12281.598} C_VEL
LIN {X 0,Y 375.929,Z 146.661,A -85,B 0,C 180,E1 -12284.731,E2 -12284.731} C_VEL
LIN {X 0,Y 375.935,Z 146.66,A -85,B 0,C 180,E1 -12288.4,E2 -12288.4} C_VEL
LIN {X 0,Y 375.973,Z 146.651,A -85,B 0,C 180,E1 -12291.73,E2 -12291.73} C_VEL
LIN {X 0,Y 375.982,Z 146.646,A -85,B 0,C 180,E1 -12295.333,E2 -12295.333} C_VEL
LIN {X 0,Y 375.983,Z 146.801,A -85,B 0,C 180,E1 -12299.051,E2 -12299.051} C_VEL
LIN {X 0,Y 378.541,Z 157.337,A -85,B 0,C 180,E1 -12301.742,E2 -12301.742} C_VEL
LIN {X 0,Y 380.358,Z 166.561,A -85,B 0,C 180,E1 -12303.97,E2 -12303.97} C_VEL
LIN {X 0,Y 380.334,Z 170.517,A -85,B 0,C 180,E1 -12304.849,E2 -12304.849} C_VEL
LIN {X 0,Y 378.866,Z 185.439,A -85,B 0,C 180,E1 -12307.996,E2 -12307.996} C_VEL
LIN {X 0,Y 382.983,Z 206.9,A -85,B 0,C 180,E1 -12308.734,E2 -12308.734} C_VEL
LIN {X 0,Y 384.861,Z 220.009,A -85,B 0,C 180,E1 -12309.127,E2 -12309.127} C_VEL
LIN {X 0,Y 383.595,Z 294.127,A -85,B 0,C 180,E1 -12310.579,E2 -12310.579} C_VEL
LIN {X 0,Y 382.817,Z 307.869,A -85,B 0,C 180,E1 -12311.051,E2 -12311.051} C_VEL
LIN {X 0,Y 382.025,Z 319.277,A -85,B 0,C 180,E1 -12311.636,E2 -12311.636} C_VEL
LIN {X 0,Y 380.96,Z 330.764,A -85,B 0,C 180,E1 -12312.417,E2 -12312.417} C_VEL
LIN {X 0,Y 379.74,Z 342.578,A -85,B 0,C 180,E1 -12313.468,E2 -12313.468} C_VEL
LIN {X 0,Y 378.576,Z 353.163,A -85,B 0,C 180,E1 -12314.66,E2 -12314.66} C_VEL
LIN {X 0,Y 377.488,Z 362.731,A -85,B 0,C 180,E1 -12315.993,E2 -12315.993} C_VEL
LIN {X 0,Y 376.532,Z 371.976,A -85,B 0,C 180,E1 -12317.605,E2 -12317.605} C_VEL
LIN {X 0,Y 375.616,Z 379.429,A -85,B 0,C 180,E1 -12319.216,E2 -12319.216} C_VEL
LIN {X 0,Y 375.123,Z 385.439,A -85,B 0,C 180,E1 -12320.836,E2 -12320.836} C_VEL
LIN {X 0,Y 374.757,Z 390.208,A -85,B 0,C 180,E1 -12322.457,E2 -12322.457} C_VEL
LIN {X 0,Y 374.58,Z 393.598,A -85,B 0,C 180,E1 -12323.939,E2 -12323.939} C_VEL
LIN {X 0,Y 374.551,Z 396.538,A -85,B 0,C 180,E1 -12325.695,E2 -12325.695} C_VEL
LIN {X 0,Y 374.492,Z 397.802,A -85,B 0,C 180,E1 -12326.772,E2 -12326.772} C_VEL
LIN {X 0,Y 374.553,Z 398.652,A -85,B 0,C 180,E1 -12327.849,E2 -12327.849} C_VEL
LIN {X 0,Y 374.626,Z 399.077,A -85,B 0,C 180,E1 -12328.925,E2 -12328.925} C_VEL
LIN {X 0,Y 374.613,Z 399.109,A -85,B 0,C 180,E1 -12330,E2 -12330} C_VEL
LIN {X 0,Y 374.628,Z 398.754,A -85,B 0,C 180,E1 -12331.075,E2 -12331.075} C_VEL
LIN {X 0,Y 374.59,Z 397.989,A -85,B 0,C 180,E1 -12332.15,E2 -12332.15} C_VEL
LIN {X 0,Y 374.56,Z 395.155,A -85,B 0,C 180,E1 -12334.304,E2 -12334.304} C_VEL
LIN {X 0,Y 374.537,Z 391.7,A -85,B 0,C 180,E1 -12335.999,E2 -12335.999} C_VEL
LIN {X 0,Y 374.723,Z 387.513,A -85,B 0,C 180,E1 -12337.544,E2 -12337.544} C_VEL
LIN {X 0,Y 374.987,Z 381.934,A -85,B 0,C 180,E1 -12339.166,E2 -12339.166} C_VEL
LIN {X 0,Y 375.459,Z 374.957,A -85,B 0,C 180,E1 -12340.788,E2 -12340.788} C_VEL
LIN {X 0,Y 376.257,Z 366.213,A -85,B 0,C 180,E1 -12342.404,E2 -12342.404} C_VEL
LIN {X 0,Y 376.973,Z 357.226,A -85,B 0,C 180,E1 -12343.751,E2 -12343.751} C_VEL
LIN {X 0,Y 377.738,Z 347.202,A -85,B 0,C 180,E1 -12344.976,E2 -12344.976} C_VEL
LIN {X 0,Y 378.642,Z 336.487,A -85,B 0,C 180,E1 -12346.027,E2 -12346.027} C_VEL
LIN {X 0,Y 379.5,Z 324.278,A -85,B 0,C 180,E1 -12346.958,E2 -12346.958} C_VEL
LIN {X 0,Y 380.331,Z 311.543,A -85,B 0,C 180,E1 -12347.682,E2 -12347.682} C_VEL
LIN {X 0,Y 380.955,Z 298.997,A -85,B 0,C 180,E1 -12348.173,E2 -12348.173} C_VEL
LIN {X 0,Y 381.31,Z 283.095,A -85,B 0,C 180,E1 -12348.538,E2 -12348.538} C_VEL
LIN {X 0,Y 382.059,Z 218.655,A -85,B 0,C 180,E1 -12349.766,E2 -12349.766} C_VEL
LIN {X 0,Y 377.627,Z 186.197,A -85,B 0,C 180,E1 -12350.619,E2 -12350.619} C_VEL
LIN {X 0,Y 379.037,Z 167.895,A -85,B 0,C 180,E1 -12354.403,E2 -12354.403} C_VEL
LIN {X 0,Y 379.17,Z 162.566,A -85,B 0,C 180,E1 -12355.527,E2 -12355.527} C_VEL
LIN {X 0,Y 376.47,Z 148.765,A -85,B 0,C 180,E1 -12358.669,E2 -12358.669} C_VEL
LIN {X 0,Y 376.003,Z 146.65,A -85,B 0,C 180,E1 -12359.191,E2 -12359.191} C_VEL
LIN {X 0,Y 375.952,Z 146.651,A -85,B 0,C 180,E1 -12362.828,E2 -12362.828} C_VEL
LIN {X 0,Y 375.959,Z 146.652,A -85,B 0,C 180,E1 -12365.415,E2 -12365.415} C_VEL
LIN {X 0,Y 375.976,Z 146.651,A -85,B 0,C 180,E1 -12368.27,E2 -12368.27} C_VEL
LIN {X 0,Y 375.936,Z 146.658,A -85,B 0,C 180,E1 -12371.6,E2 -12371.6} C_VEL
LIN {X 0,Y 375.928,Z 146.656,A -85,B 0,C 180,E1 -12375.268,E2 -12375.268} C_VEL
LIN {X 0,Y 375.935,Z 146.654,A -85,B 0,C 180,E1 -12378.399,E2 -12378.399} C_VEL
LIN {X 0,Y 375.973,Z 146.653,A -85,B 0,C 180,E1 -12381.73,E2 -12381.73} C_VEL
LIN {X 0,Y 375.98,Z 146.653,A -85,B 0,C 180,E1 -12385.332,E2 -12385.332} C_VEL
LIN {X 0,Y 375.958,Z 146.65,A -85,B 0,C 180,E1 -12388.438,E2 -12388.438} C_VEL
LIN {X 0,Y 375.996,Z 146.646,A -85,B 0,C 180,E1 -12392.141,E2 -12392.141} C_VEL
LIN {X 0,Y 376.006,Z 146.645,A -85,B 0,C 180,E1 -12394.539,E2 -12394.539} C_VEL
LIN {X 0,Y 375.958,Z 146.65,A -85,B 0,C 180,E1 -12398.045,E2 -12398.045} C_VEL
LIN {X 0,Y 376.003,Z 146.648,A -85,B 0,C 180,E1 -12401.473,E2 -12401.473} C_VEL
LIN {X 0,Y 376.058,Z 146.642,A -85,B 0,C 180,E1 -12404.832,E2 -12404.832} C_VEL
LIN {X 0,Y 376.049,Z 146.639,A -85,B 0,C 180,E1 -12408.136,E2 -12408.136} C_VEL
LIN {X 0,Y 376.173,Z 146.624,A -85,B 0,C 180,E1 -12411.968,E2 -12411.968} C_VEL
LIN {X 0,Y 376.16,Z 146.63,A -85,B 0,C 180,E1 -12414.64,E2 -12414.64} C_VEL
LIN {X 0,Y 376.352,Z 146.601,A -85,B 0,C 180,E1 -12417.859,E2 -12417.859} C_VEL
LIN {X 0,Y 376.487,Z 146.585,A -85,B 0,C 180,E1 -12420,E2 -12420} C_VEL
LIN {X 0,Y 376.187,Z 146.623,A -85,B 0,C 180,E1 -12423.213,E2 -12423.213} C_VEL
LIN {X 0,Y 376.228,Z 146.621,A -85,B 0,C 180,E1 -12426.553,E2 -12426.553} C_VEL
LIN {X 0,Y 376.118,Z 146.631,A -85,B 0,C 180,E1 -12429.681,E2 -12429.681} C_VEL
LIN {X 0,Y 376.089,Z 146.635,A -85,B 0,C 180,E1 -12433.657,E2 -12433.657} C_VEL
LIN {X 0,Y 376.043,Z 146.64,A -85,B 0,C 180,E1 -12437.607,E2 -12437.607} C_VEL
LIN {X 0,Y 375.977,Z 146.649,A -85,B 0,C 180,E1 -12440.832,E2 -12440.832} C_VEL
LIN {X 0,Y 375.988,Z 146.652,A -85,B 0,C 180,E1 -12444.282,E2 -12444.282} C_VEL
LIN {X 0,Y 376.019,Z 146.644,A -85,B 0,C 180,E1 -12446.652,E2 -12446.652} C_VEL
LIN {X 0,Y 375.963,Z 146.653,A -85,B 0,C 180,E1 -12450.313,E2 -12450.313} C_VEL
LIN {X 0,Y 375.961,Z 146.654,A -85,B 0,C 180,E1 -12454.111,E2 -12454.111} C_VEL
LIN {X 0,Y 375.952,Z 146.651,A -85,B 0,C 180,E1 -12456.741,E2 -12456.741} C_VEL
LIN {X 0,Y 375.988,Z 146.651,A -85,B 0,C 180,E1 -12459.971,E2 -12459.971} C_VEL
LIN {X 0,Y 375.929,Z 146.66,A -85,B 0,C 180,E1 -12463.766,E2 -12463.766} C_VEL
LIN {X 0,Y 375.932,Z 146.654,A -85,B 0,C 180,E1 -12466.811,E2 -12466.811} C_VEL
LIN {X 0,Y 375.959,Z 146.65,A -85,B 0,C 180,E1 -12470.537,E2 -12470.537} C_VEL
LIN {X 0,Y 375.962,Z 146.656,A -85,B 0,C 180,E1 -12473.496,E2 -12473.496} C_VEL
LIN {X 0,Y 375.958,Z 146.652,A -85,B 0,C 180,E1 -12475.889,E2 -12475.889} C_VEL
LIN {X 0,Y 375.964,Z 146.652,A -85,B 0,C 180,E1 -12479.688,E2 -12479.688} C_VEL
LIN {X 0,Y 375.995,Z 146.646,A -85,B 0,C 180,E1 -12482.141,E2 -12482.141} C_VEL
LIN {X 0,Y 376.005,Z 146.645,A -85,B 0,C 180,E1 -12484.539,E2 -12484.539} C_VEL
LIN {X 0,Y 375.957,Z 146.651,A -85,B 0,C 180,E1 -12488.046,E2 -12488.046} C_VEL
LIN {X 0,Y 376.002,Z 146.647,A -85,B 0,C 180,E1 -12491.473,E2 -12491.473} C_VEL
LIN {X 0,Y 376.058,Z 146.643,A -85,B 0,C 180,E1 -12494.833,E2 -12494.833} C_VEL
LIN {X 0,Y 376.049,Z 146.639,A -85,B 0,C 180,E1 -12498.137,E2 -12498.137} C_VEL
LIN {X 0,Y 376.173,Z 146.624,A -85,B 0,C 180,E1 -12501.968,E2 -12501.968} C_VEL
LIN {X 0,Y 376.16,Z 146.631,A -85,B 0,C 180,E1 -12504.64,E2 -12504.64} C_VEL
LIN {X 0,Y 376.307,Z 146.732,A -85,B 0,C 180,E1 -12507.558,E2 -12507.558} C_VEL
LIN {X 0,Y 377.716,Z 154.104,A -85,B 0,C 180,E1 -12509.467,E2 -12509.467} C_VEL
LIN {X 0,Y 380.306,Z 164.247,A -85,B 0,C 180,E1 -12509.802,E2 -12509.802} C_VEL
LIN {X 0,Y 382.671,Z 177.456,A -85,B 0,C 180,E1 -12510.175,E2 -12510.175} C_VEL
LIN {X 0,Y 381.312,Z 261.26,A -85,B 0,C 180,E1 -12511.783,E2 -12511.783} C_VEL
LIN {X 0,Y 380.89,Z 274.954,A -85,B 0,C 180,E1 -12512.267,E2 -12512.267} C_VEL
LIN {X 0,Y 380.413,Z 287.477,A -85,B 0,C 180,E1 -12512.93,E2 -12512.93} C_VEL
LIN {X 0,Y 379.677,Z 299.666,A -85,B 0,C 180,E1 -12513.808,E2 -12513.808} C_VEL
LIN {X 0,Y 378.853,Z 311.573,A -85,B 0,C 180,E1 -12514.922,E2 -12514.922} C_VEL
LIN {X 0,Y 377.983,Z 321.889,A -85,B 0,C 180,E1 -12516.138,E2 -12516.138} C_VEL
LIN {X 0,Y 377.153,Z 331.153,A -85,B 0,C 180,E1 -12517.495,E2 -12517.495} C_VEL
LIN {X 0,Y 376.362,Z 340.17,A -85,B 0,C 180,E1 -12519.133,E2 -12519.133} C_VEL
LIN {X 0,Y 375.776,Z 347.372,A -85,B 0,C 180,E1 -12520.779,E2 -12520.779} C_VEL
LIN {X 0,Y 375.297,Z 353.114,A -85,B 0,C 180,E1 -12522.437,E2 -12522.437} C_VEL
LIN {X 0,Y 374.964,Z 357.616,A -85,B 0,C 180,E1 -12524.103,E2 -12524.103} C_VEL
LIN {X 0,Y 374.784,Z 359.67,A -85,B 0,C 180,E1 -12525.054,E2 -12525.054} C_VEL
LIN {X 0,Y 373.992,Z 361.279,A -85,B 0,C 180,E1 -12525.916,E2 -12525.916} C_VEL
LIN {X 0,Y 370.953,Z 363.354,A -85,B 0,C 180,E1 -12527.333,E2 -12527.333} C_VEL
LIN {X 0,Y 368.462,Z 364.52,A -85,B 0,C 180,E1 -12528.494,E2 -12528.494} C_VEL
LIN {X 0,Y 367.434,Z 365.082,A -85,B 0,C 180,E1 -12529.4,E2 -12529.4} C_VEL
LIN {X 0,Y 367.37,Z 365.153,A -85,B 0,C 180,E1 -12529.708,E2 -12529.708} C_VEL
LIN {X 0,Y 367.385,Z 365.305,A -85,B 0,C 180,E1 -12531.313,E2 -12531.313} C_VEL
LIN {X 0,Y 367.583,Z 364.173,A -85,B 0,C 180,E1 -12533.403,E2 -12533.403} C_VEL
LIN {X 0,Y 367.812,Z 362.517,A -85,B 0,C 180,E1 -12534.858,E2 -12534.858} C_VEL
LIN {X 0,Y 368.222,Z 359.454,A -85,B 0,C 180,E1 -12536.663,E2 -12536.663} C_VEL
LIN {X 0,Y 368.761,Z 355.192,A -85,B 0,C 180,E1 -12538.455,E2 -12538.455} C_VEL
LIN {X 0,Y 369.456,Z 349.461,A -85,B 0,C 180,E1 -12540.272,E2 -12540.272} C_VEL
LIN {X 0,Y 370.432,Z 342.11,A -85,B 0,C 180,E1 -12542.089,E2 -12542.089} C_VEL
LIN {X 0,Y 371.466,Z 334.185,A -85,B 0,C 180,E1 -12543.648,E2 -12543.648} C_VEL
LIN {X 0,Y 372.611,Z 324.86,A -85,B 0,C 180,E1 -12545.119,E2 -12545.119} C_VEL
LIN {X 0,Y 373.785,Z 314.97,A -85,B 0,C 180,E1 -12546.379,E2 -12546.379} C_VEL
LIN {X 0,Y 374.966,Z 303.727,A -85,B 0,C 180,E1 -12547.528,E2 -12547.528} C_VEL
LIN {X 0,Y 375.974,Z 292.117,A -85,B 0,C 180,E1 -12548.448,E2 -12548.448} C_VEL
LIN {X 0,Y 376.72,Z 280.057,A -85,B 0,C 180,E1 -12549.178,E2 -12549.178} C_VEL
LIN {X 0,Y 377.389,Z 266.878,A -85,B 0,C 180,E1 -12549.732,E2 -12549.732} C_VEL
LIN {X 0,Y 377.754,Z 252.497,A -85,B 0,C 180,E1 -12550.086,E2 -12550.086} C_VEL
LIN {X 0,Y 379.195,Z 179.018,A -85,B 0,C 180,E1 -12551.526,E2 -12551.526} C_VEL
LIN {X 0,Y 377.29,Z 171.136,A -85,B 0,C 180,E1 -12551.832,E2 -12551.832} C_VEL
LIN {X 0,Y 370.633,Z 155.193,A -85,B 0,C 180,E1 -12552.709,E2 -12552.709} C_VEL
LIN {X 0,Y 368.888,Z 147.537,A -85,B 0,C 180,E1 -12554.914,E2 -12554.914} C_VEL
LIN {X 0,Y 368.869,Z 147.541,A -85,B 0,C 180,E1 -12558.176,E2 -12558.176} C_VEL
LIN {X 0,Y 368.877,Z 147.538,A -85,B 0,C 180,E1 -12561.366,E2 -12561.366} C_VEL
LIN {X 0,Y 368.931,Z 147.532,A -85,B 0,C 180,E1 -12565.146,E2 -12565.146} C_VEL
LIN {X 0,Y 368.913,Z 147.533,A -85,B 0,C 180,E1 -12569.045,E2 -12569.045} C_VEL
LIN {X 0,Y 368.907,Z 147.531,A -85,B 0,C 180,E1 -12571.558,E2 -12571.558} C_VEL
LIN {X 0,Y 368.885,Z 147.537,A -85,B 0,C 180,E1 -12575.22,E2 -12575.22} C_VEL
LIN {X 0,Y 368.884,Z 147.528,A -85,B 0,C 180,E1 -12577.602,E2 -12577.602} C_VEL
LIN {X 0,Y 368.898,Z 147.527,A -85,B 0,C 180,E1 -12581.103,E2 -12581.103} C_VEL
LIN {X 0,Y 368.921,Z 147.525,A -85,B 0,C 180,E1 -12584.532,E2 -12584.532} C_VEL
LIN {X 0,Y 369.024,Z 147.518,A -85,B 0,C 180,E1 -12586.789,E2 -12586.789} C_VEL
LIN {X 0,Y 369.057,Z 147.509,A -85,B 0,C 180,E1 -12590.132,E2 -12590.132} C_VEL
LIN {X 0,Y 369.156,Z 147.492,A -85,B 0,C 180,E1 -12593.441,E2 -12593.441} C_VEL
LIN {X 0,Y 369.296,Z 147.475,A -85,B 0,C 180,E1 -12597.819,E2 -12597.819} C_VEL
LIN {X 0,Y 369.302,Z 147.473,A -85,B 0,C 180,E1 -12602.181,E2 -12602.181} C_VEL
LIN {X 0,Y 369.16,Z 147.496,A -85,B 0,C 180,E1 -12606.559,E2 -12606.559} C_VEL
LIN {X 0,Y 369.063,Z 147.514,A -85,B 0,C 180,E1 -12609.869,E2 -12609.869} C_VEL
LIN {X 0,Y 369.039,Z 147.511,A -85,B 0,C 180,E1 -12613.772,E2 -12613.772} C_VEL
LIN {X 0,Y 368.993,Z 147.512,A -85,B 0,C 180,E1 -12617.743,E2 -12617.743} C_VEL
LIN {X 0,Y 368.912,Z 147.526,A -85,B 0,C 180,E1 -12621.221,E2 -12621.221} C_VEL
LIN {X 0,Y 368.93,Z 147.529,A -85,B 0,C 180,E1 -12624.778,E2 -12624.778} C_VEL
LIN {X 0,Y 368.899,Z 147.535,A -85,B 0,C 180,E1 -12628.793,E2 -12628.793} C_VEL
LIN {X 0,Y 368.9,Z 147.532,A -85,B 0,C 180,E1 -12632.238,E2 -12632.238} C_VEL
LIN {X 0,Y 368.931,Z 147.529,A -85,B 0,C 180,E1 -12635.001,E2 -12635.001} C_VEL
LIN {X 0,Y 368.88,Z 147.537,A -85,B 0,C 180,E1 -12638.634,E2 -12638.634} C_VEL
LIN {X 0,Y 368.874,Z 147.538,A -85,B 0,C 180,E1 -12642.008,E2 -12642.008} C_VEL
LIN {X 0,Y 368.882,Z 147.536,A -85,B 0,C 180,E1 -12645.176,E2 -12645.176} C_VEL
LIN {X 0,Y 368.884,Z 147.537,A -85,B 0,C 180,E1 -12648.177,E2 -12648.177} C_VEL
LIN {X 0,Y 368.907,Z 147.533,A -85,B 0,C 180,E1 -12651.361,E2 -12651.361} C_VEL
LIN {X 0,Y 368.939,Z 147.523,A -85,B 0,C 180,E1 -12655.146,E2 -12655.146} C_VEL
LIN {X 0,Y 368.944,Z 147.627,A -85,B 0,C 180,E1 -12658.57,E2 -12658.57} C_VEL
LIN {X 0,Y 371.647,Z 158.787,A -85,B 0,C 180,E1 -12661.499,E2 -12661.499} C_VEL
LIN {X 0,Y 373.64,Z 169.224,A -85,B 0,C 180,E1 -12664.067,E2 -12664.067} C_VEL
LIN {X 0,Y 372.643,Z 179.783,A -85,B 0,C 180,E1 -12666.373,E2 -12666.373} C_VEL
LIN {X 0,Y 372.103,Z 184.932,A -85,B 0,C 180,E1 -12667.484,E2 -12667.484} C_VEL
LIN {X 0,Y 376.155,Z 205.695,A -85,B 0,C 180,E1 -12668.228,E2 -12668.228} C_VEL
LIN {X 0,Y 378.391,Z 221.203,A -85,B 0,C 180,E1 -12668.714,E2 -12668.714} C_VEL
LIN {X 0,Y 376.999,Z 294.55,A -85,B 0,C 180,E1 -12670.185,E2 -12670.185} C_VEL
LIN {X 0,Y 376.19,Z 308.112,A -85,B 0,C 180,E1 -12670.669,E2 -12670.669} C_VEL
LIN {X 0,Y 375.328,Z 319.926,A -85,B 0,C 180,E1 -12671.297,E2 -12671.297} C_VEL
LIN {X 0,Y 374.216,Z 331.172,A -85,B 0,C 180,E1 -12672.089,E2 -12672.089} C_VEL
LIN {X 0,Y 372.947,Z 342.81,A -85,B 0,C 180,E1 -12673.158,E2 -12673.158} C_VEL
LIN {X 0,Y 371.73,Z 353.3,A -85,B 0,C 180,E1 -12674.37,E2 -12674.37} C_VEL
LIN {X 0,Y 370.582,Z 362.784,A -85,B 0,C 180,E1 -12675.727,E2 -12675.727} C_VEL
LIN {X 0,Y 369.579,Z 371.942,A -85,B 0,C 180,E1 -12677.368,E2 -12677.368} C_VEL
LIN {X 0,Y 368.601,Z 379.344,A -85,B 0,C 180,E1 -12679.008,E2 -12679.008} C_VEL
LIN {X 0,Y 368.063,Z 385.309,A -85,B 0,C 180,E1 -12680.659,E2 -12680.659} C_VEL
LIN {X 0,Y 367.69,Z 390.037,A -85,B 0,C 180,E1 -12682.311,E2 -12682.311} C_VEL
LIN {X 0,Y 367.506,Z 393.635,A -85,B 0,C 180,E1 -12683.947,E2 -12683.947} C_VEL
LIN {X 0,Y 367.455,Z 396.291,A -85,B 0,C 180,E1 -12685.612,E2 -12685.612} C_VEL
LIN {X 0,Y 367.407,Z 397.538,A -85,B 0,C 180,E1 -12686.71,E2 -12686.71} C_VEL
LIN {X 0,Y 367.452,Z 398.352,A -85,B 0,C 180,E1 -12687.808,E2 -12687.808} C_VEL
LIN {X 0,Y 367.54,Z 398.76,A -85,B 0,C 180,E1 -12688.904,E2 -12688.904} C_VEL
LIN {X 0,Y 367.547,Z 398.776,A -85,B 0,C 180,E1 -12690,E2 -12690} C_VEL
LIN {X 0,Y 367.561,Z 398.404,A -85,B 0,C 180,E1 -12691.095,E2 -12691.095} C_VEL
LIN {X 0,Y 367.491,Z 397.601,A -85,B 0,C 180,E1 -12692.192,E2 -12692.192} C_VEL
LIN {X 0,Y 367.488,Z 394.73,A -85,B 0,C 180,E1 -12694.387,E2 -12694.387} C_VEL
LIN {X 0,Y 367.462,Z 391.528,A -85,B 0,C 180,E1 -12695.987,E2 -12695.987} C_VEL
LIN {X 0,Y 367.662,Z 387.004,A -85,B 0,C 180,E1 -12697.689,E2 -12697.689} C_VEL
LIN {X 0,Y 367.946,Z 381.378,A -85,B 0,C 180,E1 -12699.343,E2 -12699.343} C_VEL
LIN {X 0,Y 368.444,Z 374.34,A -85,B 0,C 180,E1 -12700.996,E2 -12700.996} C_VEL
LIN {X 0,Y 369.266,Z 365.512,A -85,B 0,C 180,E1 -12702.643,E2 -12702.643} C_VEL
LIN {X 0,Y 370.104,Z 355.461,A -85,B 0,C 180,E1 -12704.151,E2 -12704.151} C_VEL
LIN {X 0,Y 370.945,Z 345.212,A -85,B 0,C 180,E1 -12705.381,E2 -12705.381} C_VEL
LIN {X 0,Y 371.876,Z 333.831,A -85,B 0,C 180,E1 -12706.468,E2 -12706.468} C_VEL
LIN {X 0,Y 372.741,Z 322.033,A -85,B 0,C 180,E1 -12707.346,E2 -12707.346} C_VEL
LIN {X 0,Y 373.591,Z 309.164,A -85,B 0,C 180,E1 -12708.048,E2 -12708.048} C_VEL
LIN {X 0,Y 374.198,Z 295.44,A -85,B 0,C 180,E1 -12708.549,E2 -12708.549} C_VEL
LIN {X 0,Y 375.106,Z 238.799,A -85,B 0,C 180,E1 -12709.673,E2 -12709.673} C_VEL
LIN {X 0,Y 375.218,Z 219.161,A -85,B 0,C 180,E1 -12710.06,E2 -12710.06} C_VEL
LIN {X 0,Y 370.685,Z 185.748,A -85,B 0,C 180,E1 -12710.976,E2 -12710.976} C_VEL
LIN {X 0,Y 372.075,Z 168.772,A -85,B 0,C 180,E1 -12714.554,E2 -12714.554} C_VEL
LIN {X 0,Y 372.254,Z 164.293,A -85,B 0,C 180,E1 -12715.515,E2 -12715.515} C_VEL
LIN {X 0,Y 369.913,Z 151.993,A -85,B 0,C 180,E1 -12718.358,E2 -12718.358} C_VEL
LIN {X 0,Y 368.946,Z 147.531,A -85,B 0,C 180,E1 -12719.465,E2 -12719.465} C_VEL
LIN {X 0,Y 368.9,Z 147.53,A -85,B 0,C 180,E1 -12723.043,E2 -12723.043} C_VEL
LIN {X 0,Y 368.918,Z 147.531,A -85,B 0,C 180,E1 -12726.196,E2 -12726.196} C_VEL
LIN {X 0,Y 368.905,Z 147.529,A -85,B 0,C 180,E1 -12728.953,E2 -12728.953} C_VEL
LIN {X 0,Y 368.883,Z 147.536,A -85,B 0,C 180,E1 -12732.009,E2 -12732.009} C_VEL
LIN {X 0,Y 368.881,Z 147.534,A -85,B 0,C 180,E1 -12735.176,E2 -12735.176} C_VEL
LIN {X 0,Y 368.883,Z 147.533,A -85,B 0,C 180,E1 -12738.177,E2 -12738.177} C_VEL
LIN {X 0,Y 368.907,Z 147.533,A -85,B 0,C 180,E1 -12741.36,E2 -12741.36} C_VEL
LIN {X 0,Y 368.937,Z 147.528,A -85,B 0,C 180,E1 -12745.146,E2 -12745.146} C_VEL
LIN {X 0,Y 368.929,Z 147.529,A -85,B 0,C 180,E1 -12749.046,E2 -12749.046} C_VEL
LIN {X 0,Y 368.98,Z 147.524,A -85,B 0,C 180,E1 -12751.564,E2 -12751.564} C_VEL
LIN {X 0,Y 369,Z 147.518,A -85,B 0,C 180,E1 -12754.02,E2 -12754.02} C_VEL
LIN {X 0,Y 368.925,Z 147.529,A -85,B 0,C 180,E1 -12757.604,E2 -12757.604} C_VEL
LIN {X 0,Y 368.954,Z 147.529,A -85,B 0,C 180,E1 -12761.105,E2 -12761.105} C_VEL
LIN {X 0,Y 368.997,Z 147.519,A -85,B 0,C 180,E1 -12764.535,E2 -12764.535} C_VEL
LIN {X 0,Y 369.004,Z 147.517,A -85,B 0,C 180,E1 -12767.906,E2 -12767.906} C_VEL
LIN {X 0,Y 369.091,Z 147.509,A -85,B 0,C 180,E1 -12771.238,E2 -12771.238} C_VEL
LIN {X 0,Y 369.132,Z 147.504,A -85,B 0,C 180,E1 -12774.537,E2 -12774.537} C_VEL
LIN {X 0,Y 369.317,Z 147.478,A -85,B 0,C 180,E1 -12777.819,E2 -12777.819} C_VEL
LIN {X 0,Y 369.456,Z 147.461,A -85,B 0,C 180,E1 -12780,E2 -12780} C_VEL
LIN {X 0,Y 369.318,Z 147.48,A -85,B 0,C 180,E1 -12782.181,E2 -12782.181} C_VEL
LIN {X 0,Y 369.198,Z 147.499,A -85,B 0,C 180,E1 -12786.558,E2 -12786.558} C_VEL
LIN {X 0,Y 369.067,Z 147.51,A -85,B 0,C 180,E1 -12789.868,E2 -12789.868} C_VEL
LIN {X 0,Y 369.036,Z 147.514,A -85,B 0,C 180,E1 -12793.772,E2 -12793.772} C_VEL
LIN {X 0,Y 369,Z 147.519,A -85,B 0,C 180,E1 -12797.768,E2 -12797.768} C_VEL
LIN {X 0,Y 368.909,Z 147.529,A -85,B 0,C 180,E1 -12801.221,E2 -12801.221} C_VEL
LIN {X 0,Y 368.954,Z 147.524,A -85,B 0,C 180,E1 -12804.775,E2 -12804.775} C_VEL
LIN {X 0,Y 368.962,Z 147.522,A -85,B 0,C 180,E1 -12807.203,E2 -12807.203} C_VEL
LIN {X 0,Y 368.928,Z 147.526,A -85,B 0,C 180,E1 -12810.953,E2 -12810.953} C_VEL
LIN {X 0,Y 368.928,Z 147.526,A -85,B 0,C 180,E1 -12815.001,E2 -12815.001} C_VEL
LIN {X 0,Y 368.908,Z 147.529,A -85,B 0,C 180,E1 -12818.64,E2 -12818.64} C_VEL
LIN {X 0,Y 368.88,Z 147.536,A -85,B 0,C 180,E1 -12822.009,E2 -12822.009} C_VEL
LIN {X 0,Y 368.879,Z 147.534,A -85,B 0,C 180,E1 -12825.176,E2 -12825.176} C_VEL
LIN {X 0,Y 368.881,Z 147.533,A -85,B 0,C 180,E1 -12828.178,E2 -12828.178} C_VEL
LIN {X 0,Y 368.906,Z 147.534,A -85,B 0,C 180,E1 -12831.36,E2 -12831.36} C_VEL
LIN {X 0,Y 368.935,Z 147.529,A -85,B 0,C 180,E1 -12835.147,E2 -12835.147} C_VEL
LIN {X 0,Y 368.928,Z 147.529,A -85,B 0,C 180,E1 -12839.047,E2 -12839.047} C_VEL
LIN {X 0,Y 368.979,Z 147.523,A -85,B 0,C 180,E1 -12841.564,E2 -12841.564} C_VEL
LIN {X 0,Y 368.999,Z 147.518,A -85,B 0,C 180,E1 -12844.02,E2 -12844.02} C_VEL
LIN {X 0,Y 368.924,Z 147.529,A -85,B 0,C 180,E1 -12847.605,E2 -12847.605} C_VEL
LIN {X 0,Y 368.954,Z 147.529,A -85,B 0,C 180,E1 -12851.106,E2 -12851.106} C_VEL
LIN {X 0,Y 368.996,Z 147.52,A -85,B 0,C 180,E1 -12854.535,E2 -12854.535} C_VEL
LIN {X 0,Y 369.004,Z 147.517,A -85,B 0,C 180,E1 -12857.907,E2 -12857.907} C_VEL
LIN {X 0,Y 369.09,Z 147.508,A -85,B 0,C 180,E1 -12861.238,E2 -12861.238} C_VEL
LIN {X 0,Y 369.132,Z 147.505,A -85,B 0,C 180,E1 -12864.538,E2 -12864.538} C_VEL
LIN {X 0,Y 369.274,Z 147.65,A -85,B 0,C 180,E1 -12867.341,E2 -12867.341} C_VEL
LIN {X 0,Y 370.569,Z 154.495,A -85,B 0,C 180,E1 -12869.134,E2 -12869.134} C_VEL
LIN {X 0,Y 373.469,Z 164.74,A -85,B 0,C 180,E1 -12869.483,E2 -12869.483} C_VEL
LIN {X 0,Y 375.842,Z 177.277,A -85,B 0,C 180,E1 -12869.853,E2 -12869.853} C_VEL
LIN {X 0,Y 374.488,Z 261.917,A -85,B 0,C 180,E1 -12871.512,E2 -12871.512} C_VEL
LIN {X 0,Y 374.023,Z 275.811,A -85,B 0,C 180,E1 -12872.019,E2 -12872.019} C_VEL
LIN {X 0,Y 373.481,Z 288.671,A -85,B 0,C 180,E1 -12872.725,E2 -12872.725} C_VEL
LIN {X 0,Y 372.727,Z 300.981,A -85,B 0,C 180,E1 -12873.649,E2 -12873.649} C_VEL
LIN {X 0,Y 371.908,Z 312.316,A -85,B 0,C 180,E1 -12874.743,E2 -12874.743} C_VEL
LIN {X 0,Y 371.011,Z 322.53,A -85,B 0,C 180,E1 -12875.98,E2 -12875.98} C_VEL
LIN {X 0,Y 370.144,Z 331.746,A -85,B 0,C 180,E1 -12877.364,E2 -12877.364} C_VEL
LIN {X 0,Y 369.33,Z 340.719,A -85,B 0,C 180,E1 -12879.032,E2 -12879.032} C_VEL
LIN {X 0,Y 368.719,Z 347.865,A -85,B 0,C 180,E1 -12880.71,E2 -12880.71} C_VEL
LIN {X 0,Y 368.189,Z 354.276,A -85,B 0,C 180,E1 -12882.638,E2 -12882.638} C_VEL
LIN {X 0,Y 367.826,Z 358.694,A -85,B 0,C 180,E1 -12884.382,E2 -12884.382} C_VEL
LIN {X 0,Y 367.621,Z 360.941,A -85,B 0,C 180,E1 -12885.524,E2 -12885.524} C_VEL
LIN {X 0,Y 367.466,Z 363.138,A -85,B 0,C 180,E1 -12887.006,E2 -12887.006} C_VEL
LIN {X 0,Y 367.347,Z 364.896,A -85,B 0,C 180,E1 -12888.98,E2 -12888.98} C_VEL
LIN {X 0,Y 367.37,Z 365.153,A -85,B 0,C 180,E1 -12889.708,E2 -12889.708} C_VEL
LIN {X 0,Y 366.761,Z 365.411,A -85,B 0,C 180,E1 -12890.624,E2 -12890.624} C_VEL
LIN {X 0,Y 363.974,Z 365.27,A -85,B 0,C 180,E1 -12892.118,E2 -12892.118} C_VEL
LIN {X 0,Y 361.638,Z 364.63,A -85,B 0,C 180,E1 -12893.32,E2 -12893.32} C_VEL
LIN {X 0,Y 360.661,Z 363.629,A -85,B 0,C 180,E1 -12894.396,E2 -12894.396} C_VEL
LIN {X 0,Y 360.663,Z 363.388,A -85,B 0,C 180,E1 -12894.55,E2 -12894.55} C_VEL
LIN {X 0,Y 361.088,Z 360.536,A -85,B 0,C 180,E1 -12896.451,E2 -12896.451} C_VEL
LIN {X 0,Y 361.686,Z 356.171,A -85,B 0,C 180,E1 -12898.429,E2 -12898.429} C_VEL
LIN {X 0,Y 362.411,Z 350.688,A -85,B 0,C 180,E1 -12900.279,E2 -12900.279} C_VEL
LIN {X 0,Y 363.388,Z 343.829,A -85,B 0,C 180,E1 -12902.066,E2 -12902.066} C_VEL
LIN {X 0,Y 364.422,Z 336.135,A -85,B 0,C 180,E1 -12903.673,E2 -12903.673} C_VEL
LIN {X 0,Y 365.656,Z 327.007,A -85,B 0,C 180,E1 -12905.213,E2 -12905.213} C_VEL
LIN {X 0,Y 366.793,Z 318.001,A -85,B 0,C 180,E1 -12906.44,E2 -12906.44} C_VEL
LIN {X 0,Y 368.075,Z 306.817,A -85,B 0,C 180,E1 -12907.663,E2 -12907.663} C_VEL
LIN {X 0,Y 369.305,Z 294.461,A -85,B 0,C 180,E1 -12908.717,E2 -12908.717} C_VEL
LIN {X 0,Y 370.092,Z 282.22,A -85,B 0,C 180,E1 -12909.506,E2 -12909.506} C_VEL
LIN {X 0,Y 370.801,Z 269.078,A -85,B 0,C 180,E1 -12910.1,E2 -12910.1} C_VEL
LIN {X 0,Y 371.199,Z 256.594,A -85,B 0,C 180,E1 -12910.452,E2 -12910.452} C_VEL
LIN {X 0,Y 372.772,Z 180.248,A -85,B 0,C 180,E1 -12911.974,E2 -12911.974} C_VEL
LIN {X 0,Y 371.178,Z 173.701,A -85,B 0,C 180,E1 -12912.236,E2 -12912.236} C_VEL
LIN {X 0,Y 364.206,Z 157.409,A -85,B 0,C 180,E1 -12913.142,E2 -12913.142} C_VEL
LIN {X 0,Y 363.513,Z 155.515,A -85,B 0,C 180,E1 -12913.279,E2 -12913.279} C_VEL
LIN {X 0,Y 361.827,Z 148.417,A -85,B 0,C 180,E1 -12915.44,E2 -12915.44} C_VEL
LIN {X 0,Y 361.811,Z 148.422,A -85,B 0,C 180,E1 -12918.667,E2 -12918.667} C_VEL
LIN {X 0,Y 361.843,Z 148.415,A -85,B 0,C 180,E1 -12921.572,E2 -12921.572} C_VEL
LIN {X 0,Y 361.87,Z 148.405,A -85,B 0,C 180,E1 -12924.657,E2 -12924.657} C_VEL
LIN {X 0,Y 361.837,Z 148.415,A -85,B 0,C 180,E1 -12928.371,E2 -12928.371} C_VEL
LIN {X 0,Y 361.866,Z 148.41,A -85,B 0,C 180,E1 -12930.952,E2 -12930.952} C_VEL
LIN {X 0,Y 361.86,Z 148.41,A -85,B 0,C 180,E1 -12934.705,E2 -12934.705} C_VEL
LIN {X 0,Y 361.847,Z 148.409,A -85,B 0,C 180,E1 -12938.344,E2 -12938.344} C_VEL
LIN {X 0,Y 361.896,Z 148.402,A -85,B 0,C 180,E1 -12942.098,E2 -12942.098} C_VEL
LIN {X 0,Y 361.951,Z 148.396,A -85,B 0,C 180,E1 -12946.132,E2 -12946.132} C_VEL
LIN {X 0,Y 361.993,Z 148.386,A -85,B 0,C 180,E1 -12949.937,E2 -12949.937} C_VEL
LIN {X 0,Y 362.121,Z 148.369,A -85,B 0,C 180,E1 -12953.313,E2 -12953.313} C_VEL
LIN {X 0,Y 362.258,Z 148.352,A -85,B 0,C 180,E1 -12957.777,E2 -12957.777} C_VEL
LIN {X 0,Y 362.175,Z 148.368,A -85,B 0,C 180,E1 -12961.112,E2 -12961.112} C_VEL
LIN {X 0,Y 362.265,Z 148.349,A -85,B 0,C 180,E1 -12962.224,E2 -12962.224} C_VEL
LIN {X 0,Y 362.123,Z 148.372,A -85,B 0,C 180,E1 -12966.687,E2 -12966.687} C_VEL
LIN {X 0,Y 362,Z 148.393,A -85,B 0,C 180,E1 -12970.063,E2 -12970.063} C_VEL
